LIN {X 0,Y 520.349,Z 992.129,A -85,B 0,C 180,E1 23655.766,E2 23655.766} C_VEL
LIN {X 0,Y 520.731,Z 981.899,A -85,B 0,C 180,E1 23653.265,E2 23653.265} C_VEL
LIN {X 0,Y 521.246,Z 970.85,A -85,B 0,C 180,E1 23650.972,E2 23650.972} C_VEL
LIN {X 0,Y 521.945,Z 957.785,A -85,B 0,C 180,E1 23648.66,E2 23648.66} C_VEL
LIN {X 0,Y 522.858,Z 943.405,A -85,B 0,C 180,E1 23646.447,E2 23646.447} C_VEL
LIN {X 0,Y 523.896,Z 928.063,A -85,B 0,C 180,E1 23644.403,E2 23644.403} C_VEL
LIN {X 0,Y 525.181,Z 910.163,A -85,B 0,C 180,E1 23642.325,E2 23642.325} C_VEL
LIN {X 0,Y 526.584,Z 891.955,A -85,B 0,C 180,E1 23640.485,E2 23640.485} C_VEL
LIN {X 0,Y 527.977,Z 872.898,A -85,B 0,C 180,E1 23638.832,E2 23638.832} C_VEL
LIN {X 0,Y 529.538,Z 851.806,A -85,B 0,C 180,E1 23637.256,E2 23637.256} C_VEL
LIN {X 0,Y 530.891,Z 831.896,A -85,B 0,C 180,E1 23635.994,E2 23635.994} C_VEL
LIN {X 0,Y 532.274,Z 810.352,A -85,B 0,C 180,E1 23634.853,E2 23634.853} C_VEL
LIN {X 0,Y 533.339,Z 791.103,A -85,B 0,C 180,E1 23634.01,E2 23634.01} C_VEL
LIN {X 0,Y 534.429,Z 767.307,A -85,B 0,C 180,E1 23633.184,E2 23633.184} C_VEL
LIN {X 0,Y 535.228,Z 746.145,A -85,B 0,C 180,E1 23632.64,E2 23632.64} C_VEL
LIN {X 0,Y 535.848,Z 714.251,A -85,B 0,C 180,E1 23632.088,E2 23632.088} C_VEL
LIN {X 0,Y 538.7,Z 503.39,A -85,B 0,C 180,E1 23628.756,E2 23628.756} C_VEL
LIN {X 0,Y 539.869,Z 409.939,A -85,B 0,C 180,E1 23627.231,E2 23627.231} C_VEL
LIN {X 0,Y 537.49,Z 399.108,A -85,B 0,C 180,E1 23626.805,E2 23626.805} C_VEL
LIN {X 0,Y 531.85,Z 390.278,A -85,B 0,C 180,E1 23626.056,E2 23626.056} C_VEL
LIN {X 0,Y 523.892,Z 373.784,A -85,B 0,C 180,E1 23623.835,E2 23623.835} C_VEL
LIN {X 0,Y 520.607,Z 366.647,A -85,B 0,C 180,E1 23622.814,E2 23622.814} C_VEL
LIN {X 0,Y 520.573,Z 366.184,A -85,B 0,C 180,E1 23622.24,E2 23622.24} C_VEL
LIN {X 0,Y 520.511,Z 366.188,A -85,B 0,C 180,E1 23619.054,E2 23619.054} C_VEL
LIN {X 0,Y 520.521,Z 366.183,A -85,B 0,C 180,E1 23615.593,E2 23615.593} C_VEL
LIN {X 0,Y 520.548,Z 366.206,A -85,B 0,C 180,E1 23612.323,E2 23612.323} C_VEL
LIN {X 0,Y 520.502,Z 366.203,A -85,B 0,C 180,E1 23609.078,E2 23609.078} C_VEL
LIN {X 0,Y 520.567,Z 366.201,A -85,B 0,C 180,E1 23605.849,E2 23605.849} C_VEL
LIN {X 0,Y 520.502,Z 366.206,A -85,B 0,C 180,E1 23602.593,E2 23602.593} C_VEL
LIN {X 0,Y 520.525,Z 366.208,A -85,B 0,C 180,E1 23599.175,E2 23599.175} C_VEL
LIN {X 0,Y 520.539,Z 366.208,A -85,B 0,C 180,E1 23595.942,E2 23595.942} C_VEL
LIN {X 0,Y 520.511,Z 366.206,A -85,B 0,C 180,E1 23592.649,E2 23592.649} C_VEL
LIN {X 0,Y 520.577,Z 366.201,A -85,B 0,C 180,E1 23589.396,E2 23589.396} C_VEL
LIN {X 0,Y 520.514,Z 366.205,A -85,B 0,C 180,E1 23586.175,E2 23586.175} C_VEL
LIN {X 0,Y 520.543,Z 366.199,A -85,B 0,C 180,E1 23582.752,E2 23582.752} C_VEL
LIN {X 0,Y 520.542,Z 366.207,A -85,B 0,C 180,E1 23579.559,E2 23579.559} C_VEL
LIN {X 0,Y 520.524,Z 366.203,A -85,B 0,C 180,E1 23576.145,E2 23576.145} C_VEL
LIN {X 0,Y 520.587,Z 366.197,A -85,B 0,C 180,E1 23572.828,E2 23572.828} C_VEL
LIN {X 0,Y 520.534,Z 366.206,A -85,B 0,C 180,E1 23569.485,E2 23569.485} C_VEL
LIN {X 0,Y 520.535,Z 366.202,A -85,B 0,C 180,E1 23565.993,E2 23565.993} C_VEL
LIN {X 0,Y 520.588,Z 366.199,A -85,B 0,C 180,E1 23562.642,E2 23562.642} C_VEL
LIN {X 0,Y 520.538,Z 366.205,A -85,B 0,C 180,E1 23559.283,E2 23559.283} C_VEL
LIN {X 0,Y 520.548,Z 366.2,A -85,B 0,C 180,E1 23555.822,E2 23555.822} C_VEL
LIN {X 0,Y 520.588,Z 366.199,A -85,B 0,C 180,E1 23552.427,E2 23552.427} C_VEL
LIN {X 0,Y 520.539,Z 366.203,A -85,B 0,C 180,E1 23549.145,E2 23549.145} C_VEL
LIN {X 0,Y 520.573,Z 366.197,A -85,B 0,C 180,E1 23545.752,E2 23545.752} C_VEL
LIN {X 0,Y 520.58,Z 366.2,A -85,B 0,C 180,E1 23542.3,E2 23542.3} C_VEL
LIN {X 0,Y 520.546,Z 366.2,A -85,B 0,C 180,E1 23538.935,E2 23538.935} C_VEL
LIN {X 0,Y 520.587,Z 366.201,A -85,B 0,C 180,E1 23537.815,E2 23537.815} C_VEL
LIN {X 0,Y 519.589,Z 366.322,A -85,B 0,C 180,E1 23536.968,E2 23536.968} C_VEL
LIN {X 0,Y 513.085,Z 367.141,A -85,B 0,C 180,E1 23534.524,E2 23534.524} C_VEL
LIN {X 0,Y 512.648,Z 367.189,A -85,B 0,C 180,E1 23533.965,E2 23533.965} C_VEL
LIN {X 0,Y 512.615,Z 367.191,A -85,B 0,C 180,E1 23530.474,E2 23530.474} C_VEL
LIN {X 0,Y 512.624,Z 367.189,A -85,B 0,C 180,E1 23526.898,E2 23526.898} C_VEL
LIN {X 0,Y 512.646,Z 367.172,A -85,B 0,C 180,E1 23523.408,E2 23523.408} C_VEL
LIN {X 0,Y 512.631,Z 367.178,A -85,B 0,C 180,E1 23519.949,E2 23519.949} C_VEL
LIN {X 0,Y 512.622,Z 367.192,A -85,B 0,C 180,E1 23516.4,E2 23516.4} C_VEL
LIN {X 0,Y 512.647,Z 367.191,A -85,B 0,C 180,E1 23512.955,E2 23512.955} C_VEL
LIN {X 0,Y 512.645,Z 367.193,A -85,B 0,C 180,E1 23509.359,E2 23509.359} C_VEL
LIN {X 0,Y 512.648,Z 367.36,A -85,B 0,C 180,E1 23508.032,E2 23508.032} C_VEL
LIN {X 0,Y 513.024,Z 368.847,A -85,B 0,C 180,E1 23507.813,E2 23507.813} C_VEL
LIN {X 0,Y 514.992,Z 371.888,A -85,B 0,C 180,E1 23507.522,E2 23507.522} C_VEL
LIN {X 0,Y 516.385,Z 373.399,A -85,B 0,C 180,E1 23507.333,E2 23507.333} C_VEL
LIN {X 0,Y 519.013,Z 377.291,A -85,B 0,C 180,E1 23506.963,E2 23506.963} C_VEL
LIN {X 0,Y 530.622,Z 393.994,A -85,B 0,C 180,E1 23505.404,E2 23505.404} C_VEL
LIN {X 0,Y 533.879,Z 399.167,A -85,B 0,C 180,E1 23504.979,E2 23504.979} C_VEL
LIN {X 0,Y 530.564,Z 613.236,A -85,B 0,C 180,E1 23501.524,E2 23501.524} C_VEL
LIN {X 0,Y 529.036,Z 711.437,A -85,B 0,C 180,E1 23499.944,E2 23499.944} C_VEL
LIN {X 0,Y 528.194,Z 733.986,A -85,B 0,C 180,E1 23499.396,E2 23499.396} C_VEL
LIN {X 0,Y 527.019,Z 757.223,A -85,B 0,C 180,E1 23498.623,E2 23498.623} C_VEL
LIN {X 0,Y 525.744,Z 778.536,A -85,B 0,C 180,E1 23497.702,E2 23497.702} C_VEL
LIN {X 0,Y 524.274,Z 800.078,A -85,B 0,C 180,E1 23496.567,E2 23496.567} C_VEL
LIN {X 0,Y 522.652,Z 821.532,A -85,B 0,C 180,E1 23495.21,E2 23495.21} C_VEL
LIN {X 0,Y 520.974,Z 842.55,A -85,B 0,C 180,E1 23493.628,E2 23493.628} C_VEL
LIN {X 0,Y 519.313,Z 862.459,A -85,B 0,C 180,E1 23491.872,E2 23491.872} C_VEL
LIN {X 0,Y 517.78,Z 880.735,A -85,B 0,C 180,E1 23489.997,E2 23489.997} C_VEL
LIN {X 0,Y 516.352,Z 898.567,A -85,B 0,C 180,E1 23487.888,E2 23487.888} C_VEL
LIN {X 0,Y 515.122,Z 914.905,A -85,B 0,C 180,E1 23485.655,E2 23485.655} C_VEL
LIN {X 0,Y 514.093,Z 929.824,A -85,B 0,C 180,E1 23483.296,E2 23483.296} C_VEL
LIN {X 0,Y 513.292,Z 943.254,A -85,B 0,C 180,E1 23480.806,E2 23480.806} C_VEL
LIN {X 0,Y 512.729,Z 954.794,A -85,B 0,C 180,E1 23478.296,E2 23478.296} C_VEL
LIN {X 0,Y 512.352,Z 964.036,A -85,B 0,C 180,E1 23475.878,E2 23475.878} C_VEL
LIN {X 0,Y 512.081,Z 972.48,A -85,B 0,C 180,E1 23473.201,E2 23473.201} C_VEL
LIN {X 0,Y 511.963,Z 978.61,A -85,B 0,C 180,E1 23470.725,E2 23470.725} C_VEL
LIN {X 0,Y 511.913,Z 983.402,A -85,B 0,C 180,E1 23468.09,E2 23468.09} C_VEL
LIN {X 0,Y 511.915,Z 986.412,A -85,B 0,C 180,E1 23465.531,E2 23465.531} C_VEL
LIN {X 0,Y 511.903,Z 987.824,A -85,B 0,C 180,E1 23462.926,E2 23462.926} C_VEL
LIN {X 0,Y 511.9,Z 987.73,A -85,B 0,C 180,E1 23460.511,E2 23460.511} C_VEL
LIN {X 0,Y 511.908,Z 986.022,A -85,B 0,C 180,E1 23457.962,E2 23457.962} C_VEL
LIN {X 0,Y 511.933,Z 982.695,A -85,B 0,C 180,E1 23455.362,E2 23455.362} C_VEL
LIN {X 0,Y 511.996,Z 977.795,A -85,B 0,C 180,E1 23452.823,E2 23452.823} C_VEL
LIN {X 0,Y 512.141,Z 971.297,A -85,B 0,C 180,E1 23450.284,E2 23450.284} C_VEL
LIN {X 0,Y 512.374,Z 963.32,A -85,B 0,C 180,E1 23447.831,E2 23447.831} C_VEL
LIN {X 0,Y 512.764,Z 953.763,A -85,B 0,C 180,E1 23445.376,E2 23445.376} C_VEL
LIN {X 0,Y 513.339,Z 942.306,A -85,B 0,C 180,E1 23442.913,E2 23442.913} C_VEL
LIN {X 0,Y 514.168,Z 928.617,A -85,B 0,C 180,E1 23440.411,E2 23440.411} C_VEL
LIN {X 0,Y 515.189,Z 913.932,A -85,B 0,C 180,E1 23438.11,E2 23438.11} C_VEL
LIN {X 0,Y 516.424,Z 897.762,A -85,B 0,C 180,E1 23435.92,E2 23435.92} C_VEL
LIN {X 0,Y 517.885,Z 879.526,A -85,B 0,C 180,E1 23433.782,E2 23433.782} C_VEL
LIN {X 0,Y 519.416,Z 861.022,A -85,B 0,C 180,E1 23431.904,E2 23431.904} C_VEL
LIN {X 0,Y 521.084,Z 841.323,A -85,B 0,C 180,E1 23430.181,E2 23430.181} C_VEL
LIN {X 0,Y 522.756,Z 820.167,A -85,B 0,C 180,E1 23428.605,E2 23428.605} C_VEL
LIN {X 0,Y 524.336,Z 799.285,A -85,B 0,C 180,E1 23427.297,E2 23427.297} C_VEL
LIN {X 0,Y 525.804,Z 777.515,A -85,B 0,C 180,E1 23426.16,E2 23426.16} C_VEL
LIN {X 0,Y 527.123,Z 755.205,A -85,B 0,C 180,E1 23425.214,E2 23425.214} C_VEL
LIN {X 0,Y 528.261,Z 732.587,A -85,B 0,C 180,E1 23424.473,E2 23424.473} C_VEL
LIN {X 0,Y 529.086,Z 709.622,A -85,B 0,C 180,E1 23423.929,E2 23423.929} C_VEL
LIN {X 0,Y 532.283,Z 499.238,A -85,B 0,C 180,E1 23420.56,E2 23420.56} C_VEL
LIN {X 0,Y 533.734,Z 398.668,A -85,B 0,C 180,E1 23418.906,E2 23418.906} C_VEL
LIN {X 0,Y 524.824,Z 385.59,A -85,B 0,C 180,E1 23417.734,E2 23417.734} C_VEL
LIN {X 0,Y 519.029,Z 377.339,A -85,B 0,C 180,E1 23416.94,E2 23416.94} C_VEL
LIN {X 0,Y 516.307,Z 373.278,A -85,B 0,C 180,E1 23416.554,E2 23416.554} C_VEL
LIN {X 0,Y 513.441,Z 369.804,A -85,B 0,C 180,E1 23416.154,E2 23416.154} C_VEL
LIN {X 0,Y 512.74,Z 367.777,A -85,B 0,C 180,E1 23415.96,E2 23415.96} C_VEL
LIN {X 0,Y 512.647,Z 367.178,A -85,B 0,C 180,E1 23415.614,E2 23415.614} C_VEL
LIN {X 0,Y 512.643,Z 367.188,A -85,B 0,C 180,E1 23412.046,E2 23412.046} C_VEL
LIN {X 0,Y 512.634,Z 367.194,A -85,B 0,C 180,E1 23408.525,E2 23408.525} C_VEL
LIN {X 0,Y 512.641,Z 367.184,A -85,B 0,C 180,E1 23405.036,E2 23405.036} C_VEL
LIN {X 0,Y 512.631,Z 367.193,A -85,B 0,C 180,E1 23401.565,E2 23401.565} C_VEL
LIN {X 0,Y 512.644,Z 367.19,A -85,B 0,C 180,E1 23398.1,E2 23398.1} C_VEL
LIN {X 0,Y 512.642,Z 367.186,A -85,B 0,C 180,E1 23394.516,E2 23394.516} C_VEL
LIN {X 0,Y 512.622,Z 367.191,A -85,B 0,C 180,E1 23391.137,E2 23391.137} C_VEL
LIN {X 0,Y 512.622,Z 367.194,A -85,B 0,C 180,E1 23387.611,E2 23387.611} C_VEL
LIN {X 0,Y 512.648,Z 367.191,A -85,B 0,C 180,E1 23384.154,E2 23384.154} C_VEL
LIN {X 0,Y 512.616,Z 367.192,A -85,B 0,C 180,E1 23380.746,E2 23380.746} C_VEL
LIN {X 0,Y 512.601,Z 367.193,A -85,B 0,C 180,E1 23377.282,E2 23377.282} C_VEL
LIN {X 0,Y 512.647,Z 367.187,A -85,B 0,C 180,E1 23373.971,E2 23373.971} C_VEL
LIN {X 0,Y 512.588,Z 367.189,A -85,B 0,C 180,E1 23370.686,E2 23370.686} C_VEL
LIN {X 0,Y 512.587,Z 367.199,A -85,B 0,C 180,E1 23367.162,E2 23367.162} C_VEL
LIN {X 0,Y 512.63,Z 367.19,A -85,B 0,C 180,E1 23363.854,E2 23363.854} C_VEL
LIN {X 0,Y 512.567,Z 367.202,A -85,B 0,C 180,E1 23360.512,E2 23360.512} C_VEL
LIN {X 0,Y 512.633,Z 367.461,A -85,B 0,C 180,E1 23358,E2 23358} C_VEL
LIN {X 0,Y 514.255,Z 371.158,A -85,B 0,C 180,E1 23357.421,E2 23357.421} C_VEL
LIN {X 0,Y 522.336,Z 388.024,A -85,B 0,C 180,E1 23355.063,E2 23355.063} C_VEL
LIN {X 0,Y 524.102,Z 391.266,A -85,B 0,C 180,E1 23354.714,E2 23354.714} C_VEL
LIN {X 0,Y 532.473,Z 404.496,A -85,B 0,C 180,E1 23353.596,E2 23353.596} C_VEL
LIN {X 0,Y 534.057,Z 413.512,A -85,B 0,C 180,E1 23353.272,E2 23353.272} C_VEL
LIN {X 0,Y 530.901,Z 620.252,A -85,B 0,C 180,E1 23349.935,E2 23349.935} C_VEL
LIN {X 0,Y 529.048,Z 740.56,A -85,B 0,C 180,E1 23348.004,E2 23348.004} C_VEL
LIN {X 0,Y 528.187,Z 763.41,A -85,B 0,C 180,E1 23347.452,E2 23347.452} C_VEL
LIN {X 0,Y 527.178,Z 784.187,A -85,B 0,C 180,E1 23346.778,E2 23346.778} C_VEL
LIN {X 0,Y 525.864,Z 806.34,A -85,B 0,C 180,E1 23345.849,E2 23345.849} C_VEL
LIN {X 0,Y 524.54,Z 826.536,A -85,B 0,C 180,E1 23344.815,E2 23344.815} C_VEL
LIN {X 0,Y 522.895,Z 848.102,A -85,B 0,C 180,E1 23343.483,E2 23343.483} C_VEL
LIN {X 0,Y 521.357,Z 867.974,A -85,B 0,C 180,E1 23342.042,E2 23342.042} C_VEL
LIN {X 0,Y 519.726,Z 887.242,A -85,B 0,C 180,E1 23340.398,E2 23340.398} C_VEL
LIN {X 0,Y 518.112,Z 906.765,A -85,B 0,C 180,E1 23338.47,E2 23338.47} C_VEL
LIN {X 0,Y 516.731,Z 923.638,A -85,B 0,C 180,E1 23336.553,E2 23336.553} C_VEL
LIN {X 0,Y 515.543,Z 939.127,A -85,B 0,C 180,E1 23334.524,E2 23334.524} C_VEL
LIN {X 0,Y 514.479,Z 954.204,A -85,B 0,C 180,E1 23332.273,E2 23332.273} C_VEL
LIN {X 0,Y 513.631,Z 967.075,A -85,B 0,C 180,E1 23330.039,E2 23330.039} C_VEL
LIN {X 0,Y 512.948,Z 979.793,A -85,B 0,C 180,E1 23327.471,E2 23327.471} C_VEL
LIN {X 0,Y 512.523,Z 989.518,A -85,B 0,C 180,E1 23325.157,E2 23325.157} C_VEL
LIN {X 0,Y 512.205,Z 998.524,A -85,B 0,C 180,E1 23322.571,E2 23322.571} C_VEL
LIN {X 0,Y 512.027,Z 1005.249,A -85,B 0,C 180,E1 23320.206,E2 23320.206} C_VEL
LIN {X 0,Y 511.953,Z 1010.629,A -85,B 0,C 180,E1 23317.748,E2 23317.748} C_VEL
LIN {X 0,Y 511.91,Z 1014.273,A -85,B 0,C 180,E1 23315.495,E2 23315.495} C_VEL
LIN {X 0,Y 511.89,Z 1016.917,A -85,B 0,C 180,E1 23312.914,E2 23312.914} C_VEL
LIN {X 0,Y 511.883,Z 1017.872,A -85,B 0,C 180,E1 23310.675,E2 23310.675} C_VEL
LIN {X 0,Y 511.909,Z 1017.528,A -85,B 0,C 180,E1 23308.101,E2 23308.101} C_VEL
LIN {X 0,Y 511.911,Z 1015.733,A -85,B 0,C 180,E1 23305.747,E2 23305.747} C_VEL
LIN {X 0,Y 511.925,Z 1012.5,A -85,B 0,C 180,E1 23303.274,E2 23303.274} C_VEL
LIN {X 0,Y 511.996,Z 1007.837,A -85,B 0,C 180,E1 23300.902,E2 23300.902} C_VEL
LIN {X 0,Y 512.119,Z 1001.528,A -85,B 0,C 180,E1 23298.403,E2 23298.403} C_VEL
LIN {X 0,Y 512.355,Z 993.422,A -85,B 0,C 180,E1 23295.903,E2 23295.903} C_VEL
LIN {X 0,Y 512.746,Z 983.956,A -85,B 0,C 180,E1 23293.463,E2 23293.463} C_VEL
LIN {X 0,Y 513.275,Z 973.174,A -85,B 0,C 180,E1 23291.138,E2 23291.138} C_VEL
LIN {X 0,Y 514.072,Z 959.885,A -85,B 0,C 180,E1 23288.676,E2 23288.676} C_VEL
LIN {X 0,Y 514.991,Z 946.596,A -85,B 0,C 180,E1 23286.551,E2 23286.551} C_VEL
LIN {X 0,Y 516.168,Z 930.762,A -85,B 0,C 180,E1 23284.351,E2 23284.351} C_VEL
LIN {X 0,Y 517.52,Z 914.034,A -85,B 0,C 180,E1 23282.317,E2 23282.317} C_VEL
LIN {X 0,Y 518.986,Z 896.227,A -85,B 0,C 180,E1 23280.454,E2 23280.454} C_VEL
LIN {X 0,Y 520.627,Z 876.321,A -85,B 0,C 180,E1 23278.643,E2 23278.643} C_VEL
LIN {X 0,Y 522.234,Z 856.967,A -85,B 0,C 180,E1 23277.132,E2 23277.132} C_VEL
LIN {X 0,Y 523.815,Z 835.912,A -85,B 0,C 180,E1 23275.735,E2 23275.735} C_VEL
LIN {X 0,Y 525.403,Z 814.179,A -85,B 0,C 180,E1 23274.525,E2 23274.525} C_VEL
LIN {X 0,Y 526.667,Z 793.392,A -85,B 0,C 180,E1 23273.586,E2 23273.586} C_VEL
LIN {X 0,Y 527.825,Z 771.737,A -85,B 0,C 180,E1 23272.79,E2 23272.79} C_VEL
LIN {X 0,Y 528.721,Z 749.391,A -85,B 0,C 180,E1 23272.186,E2 23272.186} C_VEL
LIN {X 0,Y 529.41,Z 723.55,A -85,B 0,C 180,E1 23271.701,E2 23271.701} C_VEL
LIN {X 0,Y 532.519,Z 513.255,A -85,B 0,C 180,E1 23268.347,E2 23268.347} C_VEL
LIN {X 0,Y 533.929,Z 411.728,A -85,B 0,C 180,E1 23266.678,E2 23266.678} C_VEL
LIN {X 0,Y 532.159,Z 403.642,A -85,B 0,C 180,E1 23266.352,E2 23266.352} C_VEL
LIN {X 0,Y 523.281,Z 389.92,A -85,B 0,C 180,E1 23265.144,E2 23265.144} C_VEL
LIN {X 0,Y 516.26,Z 375.275,A -85,B 0,C 180,E1 23263.108,E2 23263.108} C_VEL
LIN {X 0,Y 512.665,Z 367.588,A -85,B 0,C 180,E1 23261.958,E2 23261.958} C_VEL
LIN {X 0,Y 512.577,Z 367.19,A -85,B 0,C 180,E1 23261.099,E2 23261.099} C_VEL
LIN {X 0,Y 512.585,Z 367.2,A -85,B 0,C 180,E1 23257.628,E2 23257.628} C_VEL
LIN {X 0,Y 512.616,Z 367.174,A -85,B 0,C 180,E1 23254.311,E2 23254.311} C_VEL
LIN {X 0,Y 512.563,Z 367.176,A -85,B 0,C 180,E1 23250.996,E2 23250.996} C_VEL
LIN {X 0,Y 512.608,Z 367.197,A -85,B 0,C 180,E1 23247.66,E2 23247.66} C_VEL
LIN {X 0,Y 512.578,Z 367.199,A -85,B 0,C 180,E1 23244.376,E2 23244.376} C_VEL
LIN {X 0,Y 512.566,Z 367.194,A -85,B 0,C 180,E1 23240.887,E2 23240.887} C_VEL
LIN {X 0,Y 512.632,Z 367.19,A -85,B 0,C 180,E1 23237.596,E2 23237.596} C_VEL
LIN {X 0,Y 512.571,Z 367.191,A -85,B 0,C 180,E1 23234.343,E2 23234.343} C_VEL
LIN {X 0,Y 512.589,Z 367.195,A -85,B 0,C 180,E1 23230.906,E2 23230.906} C_VEL
LIN {X 0,Y 512.614,Z 367.191,A -85,B 0,C 180,E1 23227.621,E2 23227.621} C_VEL
LIN {X 0,Y 512.576,Z 367.194,A -85,B 0,C 180,E1 23224.25,E2 23224.25} C_VEL
LIN {X 0,Y 512.627,Z 367.193,A -85,B 0,C 180,E1 23220.894,E2 23220.894} C_VEL
LIN {X 0,Y 512.594,Z 367.193,A -85,B 0,C 180,E1 23217.652,E2 23217.652} C_VEL
LIN {X 0,Y 512.587,Z 367.194,A -85,B 0,C 180,E1 23214.106,E2 23214.106} C_VEL
LIN {X 0,Y 512.648,Z 367.193,A -85,B 0,C 180,E1 23210.797,E2 23210.797} C_VEL
LIN {X 0,Y 512.593,Z 367.192,A -85,B 0,C 180,E1 23207.495,E2 23207.495} C_VEL
LIN {X 0,Y 512.597,Z 367.192,A -85,B 0,C 180,E1 23203.919,E2 23203.919} C_VEL
LIN {X 0,Y 512.65,Z 367.192,A -85,B 0,C 180,E1 23200.517,E2 23200.517} C_VEL
LIN {X 0,Y 512.603,Z 367.191,A -85,B 0,C 180,E1 23197.159,E2 23197.159} C_VEL
LIN {X 0,Y 512.604,Z 367.191,A -85,B 0,C 180,E1 23193.594,E2 23193.594} C_VEL
LIN {X 0,Y 512.652,Z 367.19,A -85,B 0,C 180,E1 23190.175,E2 23190.175} C_VEL
LIN {X 0,Y 512.613,Z 367.193,A -85,B 0,C 180,E1 23186.763,E2 23186.763} C_VEL
LIN {X 0,Y 512.608,Z 367.192,A -85,B 0,C 180,E1 23183.214,E2 23183.214} C_VEL
LIN {X 0,Y 512.651,Z 367.186,A -85,B 0,C 180,E1 23179.791,E2 23179.791} C_VEL
LIN {X 0,Y 512.628,Z 367.191,A -85,B 0,C 180,E1 23176.333,E2 23176.333} C_VEL
LIN {X 0,Y 512.648,Z 367.189,A -85,B 0,C 180,E1 23173.965,E2 23173.965} C_VEL
LIN {X 0,Y 511.649,Z 367.308,A -85,B 0,C 180,E1 23173.104,E2 23173.104} C_VEL
LIN {X 0,Y 505.207,Z 368.114,A -85,B 0,C 180,E1 23170.684,E2 23170.684} C_VEL
LIN {X 0,Y 504.699,Z 368.177,A -85,B 0,C 180,E1 23170.054,E2 23170.054} C_VEL
LIN {X 0,Y 504.676,Z 368.181,A -85,B 0,C 180,E1 23166.602,E2 23166.602} C_VEL
LIN {X 0,Y 504.703,Z 368.163,A -85,B 0,C 180,E1 23163.07,E2 23163.07} C_VEL
LIN {X 0,Y 504.707,Z 368.158,A -85,B 0,C 180,E1 23159.551,E2 23159.551} C_VEL
LIN {X 0,Y 504.683,Z 368.173,A -85,B 0,C 180,E1 23156.087,E2 23156.087} C_VEL
LIN {X 0,Y 504.692,Z 368.177,A -85,B 0,C 180,E1 23152.475,E2 23152.475} C_VEL
LIN {X 0,Y 504.721,Z 368.305,A -85,B 0,C 180,E1 23148.979,E2 23148.979} C_VEL
LIN {X 0,Y 505.081,Z 369.781,A -85,B 0,C 180,E1 23148.738,E2 23148.738} C_VEL
LIN {X 0,Y 507.099,Z 372.938,A -85,B 0,C 180,E1 23148.424,E2 23148.424} C_VEL
LIN {X 0,Y 508.553,Z 374.512,A -85,B 0,C 180,E1 23148.219,E2 23148.219} C_VEL
LIN {X 0,Y 511.228,Z 378.407,A -85,B 0,C 180,E1 23147.826,E2 23147.826} C_VEL
LIN {X 0,Y 522.821,Z 394.818,A -85,B 0,C 180,E1 23146.209,E2 23146.209} C_VEL
LIN {X 0,Y 527.98,Z 402.563,A -85,B 0,C 180,E1 23145.518,E2 23145.518} C_VEL
LIN {X 0,Y 524.318,Z 618.399,A -85,B 0,C 180,E1 23142,E2 23142} C_VEL
LIN {X 0,Y 522.728,Z 711.407,A -85,B 0,C 180,E1 23140.487,E2 23140.487} C_VEL
LIN {X 0,Y 521.821,Z 734.028,A -85,B 0,C 180,E1 23139.933,E2 23139.933} C_VEL
LIN {X 0,Y 520.548,Z 757.204,A -85,B 0,C 180,E1 23139.156,E2 23139.156} C_VEL
LIN {X 0,Y 519.106,Z 779.291,A -85,B 0,C 180,E1 23138.191,E2 23138.191} C_VEL
LIN {X 0,Y 517.507,Z 800.717,A -85,B 0,C 180,E1 23137.043,E2 23137.043} C_VEL
LIN {X 0,Y 515.798,Z 821.334,A -85,B 0,C 180,E1 23135.726,E2 23135.726} C_VEL
LIN {X 0,Y 513.968,Z 842.409,A -85,B 0,C 180,E1 23134.124,E2 23134.124} C_VEL
LIN {X 0,Y 512.172,Z 861.761,A -85,B 0,C 180,E1 23132.402,E2 23132.402} C_VEL
LIN {X 0,Y 510.506,Z 880.135,A -85,B 0,C 180,E1 23130.502,E2 23130.502} C_VEL
LIN {X 0,Y 508.942,Z 897.623,A -85,B 0,C 180,E1 23128.421,E2 23128.421} C_VEL
LIN {X 0,Y 507.621,Z 913.339,A -85,B 0,C 180,E1 23126.27,E2 23126.27} C_VEL
LIN {X 0,Y 506.47,Z 928.424,A -85,B 0,C 180,E1 23123.877,E2 23123.877} C_VEL
LIN {X 0,Y 505.545,Z 942.067,A -85,B 0,C 180,E1 23121.352,E2 23121.352} C_VEL
LIN {X 0,Y 504.9,Z 953.235,A -85,B 0,C 180,E1 23118.922,E2 23118.922} C_VEL
LIN {X 0,Y 504.44,Z 963.155,A -85,B 0,C 180,E1 23116.354,E2 23116.354} C_VEL
LIN {X 0,Y 504.168,Z 971.121,A -85,B 0,C 180,E1 23113.877,E2 23113.877} C_VEL
LIN {X 0,Y 504.013,Z 977.756,A -85,B 0,C 180,E1 23111.251,E2 23111.251} C_VEL
LIN {X 0,Y 503.935,Z 982.605,A -85,B 0,C 180,E1 23108.707,E2 23108.707} C_VEL
LIN {X 0,Y 503.896,Z 985.917,A -85,B 0,C 180,E1 23106.119,E2 23106.119} C_VEL
LIN {X 0,Y 503.889,Z 987.674,A -85,B 0,C 180,E1 23103.607,E2 23103.607} C_VEL
LIN {X 0,Y 503.913,Z 987.841,A -85,B 0,C 180,E1 23101.049,E2 23101.049} C_VEL
LIN {X 0,Y 503.907,Z 986.433,A -85,B 0,C 180,E1 23098.346,E2 23098.346} C_VEL
LIN {X 0,Y 503.908,Z 983.561,A -85,B 0,C 180,E1 23095.835,E2 23095.835} C_VEL
LIN {X 0,Y 503.962,Z 979.096,A -85,B 0,C 180,E1 23093.278,E2 23093.278} C_VEL
LIN {X 0,Y 504.111,Z 972.871,A -85,B 0,C 180,E1 23090.673,E2 23090.673} C_VEL
LIN {X 0,Y 504.395,Z 964.46,A -85,B 0,C 180,E1 23087.929,E2 23087.929} C_VEL
LIN {X 0,Y 504.797,Z 955.293,A -85,B 0,C 180,E1 23085.476,E2 23085.476} C_VEL
LIN {X 0,Y 505.411,Z 943.967,A -85,B 0,C 180,E1 23082.945,E2 23082.945} C_VEL
LIN {X 0,Y 506.255,Z 931.103,A -85,B 0,C 180,E1 23080.5,E2 23080.5} C_VEL
LIN {X 0,Y 507.388,Z 916.279,A -85,B 0,C 180,E1 23078.083,E2 23078.083} C_VEL
LIN {X 0,Y 508.716,Z 900.445,A -85,B 0,C 180,E1 23075.853,E2 23075.853} C_VEL
LIN {X 0,Y 510.219,Z 883.315,A -85,B 0,C 180,E1 23073.757,E2 23073.757} C_VEL
LIN {X 0,Y 511.897,Z 864.989,A -85,B 0,C 180,E1 23071.822,E2 23071.822} C_VEL
LIN {X 0,Y 513.624,Z 845.937,A -85,B 0,C 180,E1 23070.084,E2 23070.084} C_VEL
LIN {X 0,Y 515.422,Z 825.761,A -85,B 0,C 180,E1 23068.503,E2 23068.503} C_VEL
LIN {X 0,Y 517.119,Z 805.535,A -85,B 0,C 180,E1 23067.15,E2 23067.15} C_VEL
LIN {X 0,Y 518.871,Z 783.109,A -85,B 0,C 180,E1 23065.903,E2 23065.903} C_VEL
LIN {X 0,Y 520.253,Z 761.88,A -85,B 0,C 180,E1 23064.946,E2 23064.946} C_VEL
LIN {X 0,Y 521.581,Z 738.114,A -85,B 0,C 180,E1 23064.1,E2 23064.1} C_VEL
LIN {X 0,Y 522.579,Z 715.323,A -85,B 0,C 180,E1 23063.508,E2 23063.508} C_VEL
LIN {X 0,Y 523.313,Z 682.027,A -85,B 0,C 180,E1 23062.927,E2 23062.927} C_VEL
LIN {X 0,Y 526.759,Z 472.174,A -85,B 0,C 180,E1 23059.538,E2 23059.538} C_VEL
LIN {X 0,Y 527.895,Z 402.246,A -85,B 0,C 180,E1 23058.372,E2 23058.372} C_VEL
LIN {X 0,Y 515.015,Z 383.608,A -85,B 0,C 180,E1 23056.612,E2 23056.612} C_VEL
LIN {X 0,Y 510.873,Z 378.049,A -85,B 0,C 180,E1 23056.02,E2 23056.02} C_VEL
LIN {X 0,Y 507.824,Z 373.56,A -85,B 0,C 180,E1 23055.561,E2 23055.561} C_VEL
LIN {X 0,Y 505.444,Z 370.693,A -85,B 0,C 180,E1 23055.21,E2 23055.21} C_VEL
LIN {X 0,Y 504.804,Z 368.876,A -85,B 0,C 180,E1 23055.039,E2 23055.039} C_VEL
LIN {X 0,Y 504.683,Z 368.168,A -85,B 0,C 180,E1 23054.69,E2 23054.69} C_VEL
LIN {X 0,Y 504.699,Z 368.178,A -85,B 0,C 180,E1 23051.195,E2 23051.195} C_VEL
LIN {X 0,Y 504.698,Z 368.176,A -85,B 0,C 180,E1 23047.743,E2 23047.743} C_VEL
LIN {X 0,Y 504.703,Z 368.18,A -85,B 0,C 180,E1 23044.204,E2 23044.204} C_VEL
LIN {X 0,Y 504.7,Z 368.18,A -85,B 0,C 180,E1 23040.682,E2 23040.682} C_VEL
LIN {X 0,Y 504.694,Z 368.172,A -85,B 0,C 180,E1 23037.162,E2 23037.162} C_VEL
LIN {X 0,Y 504.687,Z 368.181,A -85,B 0,C 180,E1 23033.631,E2 23033.631} C_VEL
LIN {X 0,Y 504.707,Z 368.18,A -85,B 0,C 180,E1 23030.191,E2 23030.191} C_VEL
LIN {X 0,Y 504.696,Z 368.179,A -85,B 0,C 180,E1 23026.715,E2 23026.715} C_VEL
LIN {X 0,Y 504.669,Z 368.182,A -85,B 0,C 180,E1 23023.306,E2 23023.306} C_VEL
LIN {X 0,Y 504.701,Z 368.176,A -85,B 0,C 180,E1 23019.836,E2 23019.836} C_VEL
LIN {X 0,Y 504.687,Z 368.176,A -85,B 0,C 180,E1 23016.41,E2 23016.41} C_VEL
LIN {X 0,Y 504.652,Z 368.182,A -85,B 0,C 180,E1 23013.018,E2 23013.018} C_VEL
LIN {X 0,Y 504.692,Z 368.183,A -85,B 0,C 180,E1 23009.657,E2 23009.657} C_VEL
LIN {X 0,Y 504.658,Z 368.185,A -85,B 0,C 180,E1 23006.307,E2 23006.307} C_VEL
LIN {X 0,Y 504.632,Z 368.188,A -85,B 0,C 180,E1 23002.821,E2 23002.821} C_VEL
LIN {X 0,Y 504.678,Z 368.179,A -85,B 0,C 180,E1 22999.472,E2 22999.472} C_VEL
LIN {X 0,Y 504.699,Z 368.65,A -85,B 0,C 180,E1 22998.829,E2 22998.829} C_VEL
LIN {X 0,Y 506.28,Z 372.154,A -85,B 0,C 180,E1 22998.276,E2 22998.276} C_VEL
LIN {X 0,Y 513.096,Z 386.032,A -85,B 0,C 180,E1 22996.229,E2 22996.229} C_VEL
LIN {X 0,Y 515.022,Z 389.931,A -85,B 0,C 180,E1 22995.74,E2 22995.74} C_VEL
LIN {X 0,Y 527.078,Z 408.684,A -85,B 0,C 180,E1 22994.071,E2 22994.071} C_VEL
LIN {X 0,Y 528.168,Z 415.327,A -85,B 0,C 180,E1 22993.835,E2 22993.835} C_VEL
LIN {X 0,Y 524.719,Z 623.112,A -85,B 0,C 180,E1 22990.451,E2 22990.451} C_VEL
LIN {X 0,Y 522.742,Z 740.56,A -85,B 0,C 180,E1 22988.546,E2 22988.546} C_VEL
LIN {X 0,Y 521.82,Z 763.278,A -85,B 0,C 180,E1 22987.994,E2 22987.994} C_VEL
LIN {X 0,Y 520.768,Z 783.428,A -85,B 0,C 180,E1 22987.337,E2 22987.337} C_VEL
LIN {X 0,Y 519.282,Z 806.337,A -85,B 0,C 180,E1 22986.376,E2 22986.376} C_VEL
LIN {X 0,Y 517.77,Z 827.658,A -85,B 0,C 180,E1 22985.27,E2 22985.27} C_VEL
LIN {X 0,Y 516.052,Z 848.221,A -85,B 0,C 180,E1 22983.978,E2 22983.978} C_VEL
LIN {X 0,Y 514.336,Z 868.226,A -85,B 0,C 180,E1 22982.51,E2 22982.51} C_VEL
LIN {X 0,Y 512.591,Z 887.24,A -85,B 0,C 180,E1 22980.867,E2 22980.867} C_VEL
LIN {X 0,Y 510.802,Z 906.763,A -85,B 0,C 180,E1 22978.916,E2 22978.916} C_VEL
LIN {X 0,Y 509.334,Z 923.13,A -85,B 0,C 180,E1 22977.032,E2 22977.032} C_VEL
LIN {X 0,Y 507.971,Z 939.125,A -85,B 0,C 180,E1 22974.915,E2 22974.915} C_VEL
LIN {X 0,Y 506.778,Z 954.206,A -85,B 0,C 180,E1 22972.63,E2 22972.63} C_VEL
LIN {X 0,Y 505.846,Z 967.073,A -85,B 0,C 180,E1 22970.361,E2 22970.361} C_VEL
LIN {X 0,Y 505.09,Z 979.613,A -85,B 0,C 180,E1 22967.794,E2 22967.794} C_VEL
LIN {X 0,Y 504.598,Z 989.517,A -85,B 0,C 180,E1 22965.401,E2 22965.401} C_VEL
LIN {X 0,Y 504.253,Z 998.337,A -85,B 0,C 180,E1 22962.834,E2 22962.834} C_VEL
LIN {X 0,Y 504.067,Z 1004.858,A -85,B 0,C 180,E1 22960.518,E2 22960.518} C_VEL
LIN {X 0,Y 503.967,Z 1010.629,A -85,B 0,C 180,E1 22957.871,E2 22957.871} C_VEL
LIN {X 0,Y 503.912,Z 1014.432,A -85,B 0,C 180,E1 22955.468,E2 22955.468} C_VEL
LIN {X 0,Y 503.895,Z 1016.985,A -85,B 0,C 180,E1 22952.847,E2 22952.847} C_VEL
LIN {X 0,Y 503.884,Z 1017.894,A -85,B 0,C 180,E1 22950.572,E2 22950.572} C_VEL
LIN {X 0,Y 503.914,Z 1017.394,A -85,B 0,C 180,E1 22947.843,E2 22947.843} C_VEL
LIN {X 0,Y 503.905,Z 1015.505,A -85,B 0,C 180,E1 22945.451,E2 22945.451} C_VEL
LIN {X 0,Y 503.919,Z 1011.807,A -85,B 0,C 180,E1 22942.782,E2 22942.782} C_VEL
LIN {X 0,Y 504,Z 1007.327,A -85,B 0,C 180,E1 22940.526,E2 22940.526} C_VEL
LIN {X 0,Y 504.182,Z 1000.48,A -85,B 0,C 180,E1 22937.869,E2 22937.869} C_VEL
LIN {X 0,Y 504.445,Z 992.949,A -85,B 0,C 180,E1 22935.542,E2 22935.542} C_VEL
LIN {X 0,Y 504.913,Z 982.926,A -85,B 0,C 180,E1 22932.962,E2 22932.962} C_VEL
LIN {X 0,Y 505.539,Z 972.015,A -85,B 0,C 180,E1 22930.598,E2 22930.598} C_VEL
LIN {X 0,Y 506.454,Z 958.482,A -85,B 0,C 180,E1 22928.096,E2 22928.096} C_VEL
LIN {X 0,Y 507.573,Z 944.064,A -85,B 0,C 180,E1 22925.79,E2 22925.79} C_VEL
LIN {X 0,Y 508.88,Z 928.361,A -85,B 0,C 180,E1 22923.631,E2 22923.631} C_VEL
LIN {X 0,Y 510.5,Z 910.161,A -85,B 0,C 180,E1 22921.457,E2 22921.457} C_VEL
LIN {X 0,Y 512.149,Z 892.227,A -85,B 0,C 180,E1 22919.595,E2 22919.595} C_VEL
LIN {X 0,Y 513.852,Z 873.379,A -85,B 0,C 180,E1 22917.918,E2 22917.918} C_VEL
LIN {X 0,Y 515.614,Z 853.592,A -85,B 0,C 180,E1 22916.389,E2 22916.389} C_VEL
LIN {X 0,Y 517.226,Z 833.899,A -85,B 0,C 180,E1 22915.102,E2 22915.102} C_VEL
LIN {X 0,Y 518.954,Z 811.631,A -85,B 0,C 180,E1 22913.88,E2 22913.88} C_VEL
LIN {X 0,Y 520.292,Z 791.097,A -85,B 0,C 180,E1 22912.96,E2 22912.96} C_VEL
LIN {X 0,Y 521.624,Z 767.185,A -85,B 0,C 180,E1 22912.119,E2 22912.119} C_VEL
LIN {X 0,Y 522.526,Z 746.63,A -85,B 0,C 180,E1 22911.582,E2 22911.582} C_VEL
LIN {X 0,Y 523.263,Z 715.28,A -85,B 0,C 180,E1 22911.024,E2 22911.024} C_VEL
LIN {X 0,Y 526.659,Z 504.774,A -85,B 0,C 180,E1 22907.633,E2 22907.633} C_VEL
LIN {X 0,Y 528.066,Z 413.605,A -85,B 0,C 180,E1 22906.117,E2 22906.117} C_VEL
LIN {X 0,Y 526.806,Z 408.028,A -85,B 0,C 180,E1 22905.881,E2 22905.881} C_VEL
LIN {X 0,Y 514.848,Z 389.549,A -85,B 0,C 180,E1 22904.202,E2 22904.202} C_VEL
LIN {X 0,Y 507.964,Z 375.562,A -85,B 0,C 180,E1 22902.16,E2 22902.16} C_VEL
LIN {X 0,Y 506.09,Z 371.882,A -85,B 0,C 180,E1 22901.591,E2 22901.591} C_VEL
LIN {X 0,Y 504.674,Z 368.414,A -85,B 0,C 180,E1 22901.022,E2 22901.022} C_VEL
LIN {X 0,Y 504.695,Z 368.171,A -85,B 0,C 180,E1 22898.149,E2 22898.149} C_VEL
LIN {X 0,Y 504.634,Z 368.159,A -85,B 0,C 180,E1 22894.794,E2 22894.794} C_VEL
LIN {X 0,Y 504.629,Z 368.166,A -85,B 0,C 180,E1 22891.273,E2 22891.273} C_VEL
LIN {X 0,Y 504.701,Z 368.181,A -85,B 0,C 180,E1 22887.936,E2 22887.936} C_VEL
LIN {X 0,Y 504.628,Z 368.188,A -85,B 0,C 180,E1 22884.584,E2 22884.584} C_VEL
LIN {X 0,Y 504.633,Z 368.183,A -85,B 0,C 180,E1 22881.015,E2 22881.015} C_VEL
LIN {X 0,Y 504.692,Z 368.178,A -85,B 0,C 180,E1 22877.644,E2 22877.644} C_VEL
LIN {X 0,Y 504.633,Z 368.18,A -85,B 0,C 180,E1 22874.339,E2 22874.339} C_VEL
LIN {X 0,Y 504.646,Z 368.184,A -85,B 0,C 180,E1 22870.849,E2 22870.849} C_VEL
LIN {X 0,Y 504.688,Z 368.18,A -85,B 0,C 180,E1 22867.513,E2 22867.513} C_VEL
LIN {X 0,Y 504.639,Z 368.184,A -85,B 0,C 180,E1 22864.09,E2 22864.09} C_VEL
LIN {X 0,Y 504.656,Z 368.183,A -85,B 0,C 180,E1 22860.567,E2 22860.567} C_VEL
LIN {X 0,Y 504.687,Z 368.183,A -85,B 0,C 180,E1 22857.274,E2 22857.274} C_VEL
LIN {X 0,Y 504.646,Z 368.184,A -85,B 0,C 180,E1 22853.858,E2 22853.858} C_VEL
LIN {X 0,Y 504.677,Z 368.181,A -85,B 0,C 180,E1 22850.42,E2 22850.42} C_VEL
LIN {X 0,Y 504.686,Z 368.182,A -85,B 0,C 180,E1 22847.063,E2 22847.063} C_VEL
LIN {X 0,Y 504.653,Z 368.182,A -85,B 0,C 180,E1 22843.659,E2 22843.659} C_VEL
LIN {X 0,Y 504.691,Z 368.18,A -85,B 0,C 180,E1 22840.197,E2 22840.197} C_VEL
LIN {X 0,Y 504.69,Z 368.182,A -85,B 0,C 180,E1 22836.781,E2 22836.781} C_VEL
LIN {X 0,Y 504.661,Z 368.181,A -85,B 0,C 180,E1 22833.31,E2 22833.31} C_VEL
LIN {X 0,Y 504.7,Z 368.178,A -85,B 0,C 180,E1 22829.919,E2 22829.919} C_VEL
LIN {X 0,Y 504.699,Z 368.184,A -85,B 0,C 180,E1 22826.445,E2 22826.445} C_VEL
LIN {X 0,Y 504.667,Z 368.182,A -85,B 0,C 180,E1 22822.965,E2 22822.965} C_VEL
LIN {X 0,Y 504.693,Z 368.174,A -85,B 0,C 180,E1 22819.472,E2 22819.472} C_VEL
LIN {X 0,Y 504.709,Z 368.175,A -85,B 0,C 180,E1 22815.944,E2 22815.944} C_VEL
LIN {X 0,Y 504.676,Z 368.176,A -85,B 0,C 180,E1 22812.493,E2 22812.493} C_VEL
LIN {X 0,Y 504.699,Z 368.177,A -85,B 0,C 180,E1 22810.054,E2 22810.054} C_VEL
LIN {X 0,Y 503.731,Z 368.302,A -85,B 0,C 180,E1 22809.179,E2 22809.179} C_VEL
LIN {X 0,Y 497.265,Z 369.111,A -85,B 0,C 180,E1 22806.721,E2 22806.721} C_VEL
LIN {X 0,Y 496.753,Z 369.172,A -85,B 0,C 180,E1 22806.08,E2 22806.08} C_VEL
LIN {X 0,Y 496.74,Z 369.163,A -85,B 0,C 180,E1 22802.5,E2 22802.5} C_VEL
LIN {X 0,Y 496.766,Z 369.144,A -85,B 0,C 180,E1 22799.012,E2 22799.012} C_VEL
LIN {X 0,Y 496.766,Z 369.147,A -85,B 0,C 180,E1 22795.509,E2 22795.509} C_VEL
LIN {X 0,Y 496.744,Z 369.154,A -85,B 0,C 180,E1 22791.982,E2 22791.982} C_VEL
LIN {X 0,Y 496.764,Z 369.284,A -85,B 0,C 180,E1 22789.955,E2 22789.955} C_VEL
LIN {X 0,Y 497.118,Z 370.749,A -85,B 0,C 180,E1 22789.707,E2 22789.707} C_VEL
LIN {X 0,Y 499.09,Z 373.88,A -85,B 0,C 180,E1 22789.386,E2 22789.386} C_VEL
LIN {X 0,Y 500.711,Z 375.549,A -85,B 0,C 180,E1 22789.149,E2 22789.149} C_VEL
LIN {X 0,Y 503.45,Z 379.533,A -85,B 0,C 180,E1 22788.729,E2 22788.729} C_VEL
LIN {X 0,Y 512.332,Z 391.907,A -85,B 0,C 180,E1 22787.429,E2 22787.429} C_VEL
LIN {X 0,Y 522.132,Z 406.185,A -85,B 0,C 180,E1 22786.067,E2 22786.067} C_VEL
LIN {X 0,Y 518.078,Z 624.715,A -85,B 0,C 180,E1 22782.467,E2 22782.467} C_VEL
LIN {X 0,Y 516.467,Z 711.379,A -85,B 0,C 180,E1 22781.042,E2 22781.042} C_VEL
LIN {X 0,Y 515.492,Z 734.051,A -85,B 0,C 180,E1 22780.484,E2 22780.484} C_VEL
LIN {X 0,Y 514.161,Z 756.616,A -85,B 0,C 180,E1 22779.722,E2 22779.722} C_VEL
LIN {X 0,Y 512.583,Z 778.901,A -85,B 0,C 180,E1 22778.748,E2 22778.748} C_VEL
LIN {X 0,Y 510.858,Z 800.427,A -85,B 0,C 180,E1 22777.588,E2 22777.588} C_VEL
LIN {X 0,Y 509.003,Z 821.123,A -85,B 0,C 180,E1 22776.255,E2 22776.255} C_VEL
LIN {X 0,Y 507.001,Z 842.269,A -85,B 0,C 180,E1 22774.634,E2 22774.634} C_VEL
LIN {X 0,Y 505.044,Z 861.645,A -85,B 0,C 180,E1 22772.89,E2 22772.89} C_VEL
LIN {X 0,Y 503.263,Z 879.541,A -85,B 0,C 180,E1 22771.021,E2 22771.021} C_VEL
LIN {X 0,Y 501.485,Z 897.558,A -85,B 0,C 180,E1 22768.854,E2 22768.854} C_VEL
LIN {X 0,Y 500.042,Z 913.276,A -85,B 0,C 180,E1 22766.672,E2 22766.672} C_VEL
LIN {X 0,Y 498.812,Z 927.695,A -85,B 0,C 180,E1 22764.36,E2 22764.36} C_VEL
LIN {X 0,Y 497.774,Z 941.447,A -85,B 0,C 180,E1 22761.798,E2 22761.798} C_VEL
LIN {X 0,Y 497.013,Z 953.174,A -85,B 0,C 180,E1 22759.214,E2 22759.214} C_VEL
LIN {X 0,Y 496.499,Z 963.198,A -85,B 0,C 180,E1 22756.577,E2 22756.577} C_VEL
LIN {X 0,Y 496.188,Z 971.346,A -85,B 0,C 180,E1 22753.987,E2 22753.987} C_VEL
LIN {X 0,Y 496.024,Z 977.904,A -85,B 0,C 180,E1 22751.336,E2 22751.336} C_VEL
LIN {X 0,Y 495.937,Z 982.85,A -85,B 0,C 180,E1 22748.661,E2 22748.661} C_VEL
LIN {X 0,Y 495.905,Z 986.129,A -85,B 0,C 180,E1 22745.963,E2 22745.963} C_VEL
LIN {X 0,Y 495.906,Z 987.763,A -85,B 0,C 180,E1 22743.278,E2 22743.278} C_VEL
LIN {X 0,Y 495.918,Z 987.795,A -85,B 0,C 180,E1 22740.794,E2 22740.794} C_VEL
LIN {X 0,Y 495.911,Z 986.252,A -85,B 0,C 180,E1 22738.085,E2 22738.085} C_VEL
LIN {X 0,Y 495.929,Z 983.225,A -85,B 0,C 180,E1 22735.488,E2 22735.488} C_VEL
LIN {X 0,Y 496.011,Z 978.34,A -85,B 0,C 180,E1 22732.773,E2 22732.773} C_VEL
LIN {X 0,Y 496.166,Z 972.345,A -85,B 0,C 180,E1 22730.294,E2 22730.294} C_VEL
LIN {X 0,Y 496.466,Z 964.008,A -85,B 0,C 180,E1 22727.569,E2 22727.569} C_VEL
LIN {X 0,Y 496.94,Z 954.753,A -85,B 0,C 180,E1 22725.069,E2 22725.069} C_VEL
LIN {X 0,Y 497.66,Z 943.124,A -85,B 0,C 180,E1 22722.46,E2 22722.46} C_VEL
LIN {X 0,Y 498.651,Z 929.788,A -85,B 0,C 180,E1 22719.915,E2 22719.915} C_VEL
LIN {X 0,Y 499.879,Z 915.029,A -85,B 0,C 180,E1 22717.506,E2 22717.506} C_VEL
LIN {X 0,Y 501.392,Z 898.602,A -85,B 0,C 180,E1 22715.192,E2 22715.192} C_VEL
LIN {X 0,Y 503.12,Z 881.085,A -85,B 0,C 180,E1 22713.061,E2 22713.061} C_VEL
LIN {X 0,Y 504.949,Z 862.697,A -85,B 0,C 180,E1 22711.119,E2 22711.119} C_VEL
LIN {X 0,Y 506.934,Z 842.907,A -85,B 0,C 180,E1 22709.33,E2 22709.33} C_VEL
LIN {X 0,Y 508.859,Z 822.505,A -85,B 0,C 180,E1 22707.755,E2 22707.755} C_VEL
LIN {X 0,Y 510.771,Z 801.449,A -85,B 0,C 180,E1 22706.383,E2 22706.383} C_VEL
LIN {X 0,Y 512.489,Z 780.375,A -85,B 0,C 180,E1 22705.233,E2 22705.233} C_VEL
LIN {X 0,Y 514.097,Z 757.712,A -85,B 0,C 180,E1 22704.229,E2 22704.229} C_VEL
LIN {X 0,Y 515.435,Z 734.943,A -85,B 0,C 180,E1 22703.453,E2 22703.453} C_VEL
LIN {X 0,Y 516.414,Z 712.697,A -85,B 0,C 180,E1 22702.896,E2 22702.896} C_VEL
LIN {X 0,Y 517.345,Z 667.633,A -85,B 0,C 180,E1 22702.137,E2 22702.137} C_VEL
LIN {X 0,Y 521.149,Z 457.427,A -85,B 0,C 180,E1 22698.697,E2 22698.697} C_VEL
LIN {X 0,Y 522.03,Z 405.932,A -85,B 0,C 180,E1 22697.82,E2 22697.82} C_VEL
LIN {X 0,Y 510.672,Z 389.477,A -85,B 0,C 180,E1 22696.23,E2 22696.23} C_VEL
LIN {X 0,Y 503.537,Z 379.61,A -85,B 0,C 180,E1 22695.163,E2 22695.163} C_VEL
LIN {X 0,Y 500.777,Z 375.667,A -85,B 0,C 180,E1 22694.734,E2 22694.734} C_VEL
LIN {X 0,Y 499.721,Z 374.429,A -85,B 0,C 180,E1 22694.573,E2 22694.573} C_VEL
LIN {X 0,Y 497.484,Z 371.592,A -85,B 0,C 180,E1 22694.224,E2 22694.224} C_VEL
LIN {X 0,Y 496.937,Z 370.061,A -85,B 0,C 180,E1 22694.091,E2 22694.091} C_VEL
LIN {X 0,Y 496.77,Z 369.196,A -85,B 0,C 180,E1 22693.799,E2 22693.799} C_VEL
LIN {X 0,Y 496.766,Z 369.167,A -85,B 0,C 180,E1 22690.183,E2 22690.183} C_VEL
LIN {X 0,Y 496.754,Z 369.168,A -85,B 0,C 180,E1 22686.705,E2 22686.705} C_VEL
LIN {X 0,Y 496.764,Z 369.165,A -85,B 0,C 180,E1 22683.116,E2 22683.116} C_VEL
LIN {X 0,Y 496.75,Z 369.167,A -85,B 0,C 180,E1 22679.539,E2 22679.539} C_VEL
LIN {X 0,Y 496.761,Z 369.172,A -85,B 0,C 180,E1 22675.961,E2 22675.961} C_VEL
LIN {X 0,Y 496.769,Z 369.17,A -85,B 0,C 180,E1 22672.367,E2 22672.367} C_VEL
LIN {X 0,Y 496.752,Z 369.167,A -85,B 0,C 180,E1 22668.859,E2 22668.859} C_VEL
LIN {X 0,Y 496.733,Z 369.172,A -85,B 0,C 180,E1 22665.309,E2 22665.309} C_VEL
LIN {X 0,Y 496.761,Z 369.171,A -85,B 0,C 180,E1 22661.813,E2 22661.813} C_VEL
LIN {X 0,Y 496.767,Z 369.165,A -85,B 0,C 180,E1 22658.264,E2 22658.264} C_VEL
LIN {X 0,Y 496.717,Z 369.174,A -85,B 0,C 180,E1 22654.867,E2 22654.867} C_VEL
LIN {X 0,Y 496.726,Z 369.168,A -85,B 0,C 180,E1 22651.36,E2 22651.36} C_VEL
LIN {X 0,Y 496.761,Z 369.164,A -85,B 0,C 180,E1 22647.93,E2 22647.93} C_VEL
LIN {X 0,Y 496.699,Z 369.178,A -85,B 0,C 180,E1 22644.568,E2 22644.568} C_VEL
LIN {X 0,Y 496.692,Z 369.174,A -85,B 0,C 180,E1 22640.945,E2 22640.945} C_VEL
LIN {X 0,Y 496.784,Z 369.454,A -85,B 0,C 180,E1 22639.796,E2 22639.796} C_VEL
LIN {X 0,Y 498.423,Z 373.231,A -85,B 0,C 180,E1 22639.159,E2 22639.159} C_VEL
LIN {X 0,Y 503.937,Z 384.485,A -85,B 0,C 180,E1 22637.424,E2 22637.424} C_VEL
LIN {X 0,Y 506.331,Z 389.138,A -85,B 0,C 180,E1 22636.773,E2 22636.773} C_VEL
LIN {X 0,Y 521.685,Z 412.757,A -85,B 0,C 180,E1 22634.562,E2 22634.562} C_VEL
LIN {X 0,Y 522.328,Z 417.339,A -85,B 0,C 180,E1 22634.407,E2 22634.407} C_VEL
LIN {X 0,Y 518.509,Z 625.8,A -85,B 0,C 180,E1 22630.972,E2 22630.972} C_VEL
LIN {X 0,Y 516.495,Z 739.954,A -85,B 0,C 180,E1 22629.113,E2 22629.113} C_VEL
LIN {X 0,Y 515.508,Z 763.015,A -85,B 0,C 180,E1 22628.553,E2 22628.553} C_VEL
LIN {X 0,Y 514.401,Z 782.775,A -85,B 0,C 180,E1 22627.907,E2 22627.907} C_VEL
LIN {X 0,Y 512.762,Z 806.22,A -85,B 0,C 180,E1 22626.92,E2 22626.92} C_VEL
LIN {X 0,Y 511.111,Z 827.661,A -85,B 0,C 180,E1 22625.8,E2 22625.8} C_VEL
LIN {X 0,Y 509.273,Z 848.096,A -85,B 0,C 180,E1 22624.503,E2 22624.503} C_VEL
LIN {X 0,Y 507.387,Z 868.15,A -85,B 0,C 180,E1 22623.019,E2 22623.019} C_VEL
LIN {X 0,Y 505.493,Z 887.237,A -85,B 0,C 180,E1 22621.349,E2 22621.349} C_VEL
LIN {X 0,Y 503.525,Z 906.762,A -85,B 0,C 180,E1 22619.374,E2 22619.374} C_VEL
LIN {X 0,Y 501.933,Z 923.13,A -85,B 0,C 180,E1 22617.464,E2 22617.464} C_VEL
LIN {X 0,Y 500.416,Z 939.123,A -85,B 0,C 180,E1 22615.317,E2 22615.317} C_VEL
LIN {X 0,Y 499.166,Z 953.49,A -85,B 0,C 180,E1 22613.119,E2 22613.119} C_VEL
LIN {X 0,Y 498.079,Z 967.072,A -85,B 0,C 180,E1 22610.693,E2 22610.693} C_VEL
LIN {X 0,Y 497.254,Z 979.275,A -85,B 0,C 180,E1 22608.163,E2 22608.163} C_VEL
LIN {X 0,Y 496.697,Z 989.057,A -85,B 0,C 180,E1 22605.772,E2 22605.772} C_VEL
LIN {X 0,Y 496.295,Z 998.338,A -85,B 0,C 180,E1 22603.044,E2 22603.044} C_VEL
LIN {X 0,Y 496.085,Z 1004.858,A -85,B 0,C 180,E1 22600.689,E2 22600.689} C_VEL
LIN {X 0,Y 495.974,Z 1010.629,A -85,B 0,C 180,E1 22597.999,E2 22597.999} C_VEL
LIN {X 0,Y 495.911,Z 1014.432,A -85,B 0,C 180,E1 22595.557,E2 22595.557} C_VEL
LIN {X 0,Y 495.892,Z 1016.984,A -85,B 0,C 180,E1 22592.893,E2 22592.893} C_VEL
LIN {X 0,Y 495.884,Z 1017.894,A -85,B 0,C 180,E1 22590.581,E2 22590.581} C_VEL
LIN {X 0,Y 495.914,Z 1017.394,A -85,B 0,C 180,E1 22587.808,E2 22587.808} C_VEL
LIN {X 0,Y 495.906,Z 1015.505,A -85,B 0,C 180,E1 22585.378,E2 22585.378} C_VEL
LIN {X 0,Y 495.924,Z 1011.881,A -85,B 0,C 180,E1 22582.707,E2 22582.707} C_VEL
LIN {X 0,Y 496.008,Z 1007.327,A -85,B 0,C 180,E1 22580.372,E2 22580.372} C_VEL
LIN {X 0,Y 496.208,Z 1000.743,A -85,B 0,C 180,E1 22577.76,E2 22577.76} C_VEL
LIN {X 0,Y 496.518,Z 992.951,A -85,B 0,C 180,E1 22575.306,E2 22575.306} C_VEL
LIN {X 0,Y 497.063,Z 982.41,A -85,B 0,C 180,E1 22572.564,E2 22572.564} C_VEL
LIN {X 0,Y 497.777,Z 971.436,A -85,B 0,C 180,E1 22570.16,E2 22570.16} C_VEL
LIN {X 0,Y 498.75,Z 958.48,A -85,B 0,C 180,E1 22567.74,E2 22567.74} C_VEL
LIN {X 0,Y 499.969,Z 944.245,A -85,B 0,C 180,E1 22565.425,E2 22565.425} C_VEL
LIN {X 0,Y 501.403,Z 928.445,A -85,B 0,C 180,E1 22563.218,E2 22563.218} C_VEL
LIN {X 0,Y 503.197,Z 910.159,A -85,B 0,C 180,E1 22561.004,E2 22561.004} C_VEL
LIN {X 0,Y 505.032,Z 891.955,A -85,B 0,C 180,E1 22559.091,E2 22559.091} C_VEL
LIN {X 0,Y 506.916,Z 872.826,A -85,B 0,C 180,E1 22557.375,E2 22557.375} C_VEL
LIN {X 0,Y 508.848,Z 852.705,A -85,B 0,C 180,E1 22555.813,E2 22555.813} C_VEL
LIN {X 0,Y 510.623,Z 832.991,A -85,B 0,C 180,E1 22554.521,E2 22554.521} C_VEL
LIN {X 0,Y 512.467,Z 810.472,A -85,B 0,C 180,E1 22553.286,E2 22553.286} C_VEL
LIN {X 0,Y 513.939,Z 789.615,A -85,B 0,C 180,E1 22552.353,E2 22552.353} C_VEL
LIN {X 0,Y 515.316,Z 766.662,A -85,B 0,C 180,E1 22551.554,E2 22551.554} C_VEL
LIN {X 0,Y 516.264,Z 746.467,A -85,B 0,C 180,E1 22551.025,E2 22551.025} C_VEL
LIN {X 0,Y 517.039,Z 715.438,A -85,B 0,C 180,E1 22550.468,E2 22550.468} C_VEL
LIN {X 0,Y 520.686,Z 506.52,A -85,B 0,C 180,E1 22547.07,E2 22547.07} C_VEL
LIN {X 0,Y 522.241,Z 415.425,A -85,B 0,C 180,E1 22545.539,E2 22545.539} C_VEL
LIN {X 0,Y 521.413,Z 412.278,A -85,B 0,C 180,E1 22545.39,E2 22545.39} C_VEL
LIN {X 0,Y 506.262,Z 389.027,A -85,B 0,C 180,E1 22543.182,E2 22543.182} C_VEL
LIN {X 0,Y 500.427,Z 377.299,A -85,B 0,C 180,E1 22541.402,E2 22541.402} C_VEL
LIN {X 0,Y 496.837,Z 369.662,A -85,B 0,C 180,E1 22540.176,E2 22540.176} C_VEL
LIN {X 0,Y 496.698,Z 369.143,A -85,B 0,C 180,E1 22539.566,E2 22539.566} C_VEL
LIN {X 0,Y 496.752,Z 369.144,A -85,B 0,C 180,E1 22536.193,E2 22536.193} C_VEL
LIN {X 0,Y 496.699,Z 369.178,A -85,B 0,C 180,E1 22532.718,E2 22532.718} C_VEL
LIN {X 0,Y 496.687,Z 369.16,A -85,B 0,C 180,E1 22529.154,E2 22529.154} C_VEL
LIN {X 0,Y 496.748,Z 369.166,A -85,B 0,C 180,E1 22525.891,E2 22525.891} C_VEL
LIN {X 0,Y 496.69,Z 369.173,A -85,B 0,C 180,E1 22522.487,E2 22522.487} C_VEL
LIN {X 0,Y 496.694,Z 369.175,A -85,B 0,C 180,E1 22518.91,E2 22518.91} C_VEL
LIN {X 0,Y 496.761,Z 369.167,A -85,B 0,C 180,E1 22515.527,E2 22515.527} C_VEL
LIN {X 0,Y 496.699,Z 369.173,A -85,B 0,C 180,E1 22512.202,E2 22512.202} C_VEL
LIN {X 0,Y 496.699,Z 369.167,A -85,B 0,C 180,E1 22508.566,E2 22508.566} C_VEL
LIN {X 0,Y 496.759,Z 369.165,A -85,B 0,C 180,E1 22505.196,E2 22505.196} C_VEL
LIN {X 0,Y 496.716,Z 369.167,A -85,B 0,C 180,E1 22501.73,E2 22501.73} C_VEL
LIN {X 0,Y 496.707,Z 369.17,A -85,B 0,C 180,E1 22498.269,E2 22498.269} C_VEL
LIN {X 0,Y 496.759,Z 369.168,A -85,B 0,C 180,E1 22494.803,E2 22494.803} C_VEL
LIN {X 0,Y 496.723,Z 369.166,A -85,B 0,C 180,E1 22491.433,E2 22491.433} C_VEL
LIN {X 0,Y 496.713,Z 369.169,A -85,B 0,C 180,E1 22487.915,E2 22487.915} C_VEL
LIN {X 0,Y 496.765,Z 369.168,A -85,B 0,C 180,E1 22484.472,E2 22484.472} C_VEL
LIN {X 0,Y 496.742,Z 369.166,A -85,B 0,C 180,E1 22480.969,E2 22480.969} C_VEL
LIN {X 0,Y 496.719,Z 369.168,A -85,B 0,C 180,E1 22477.493,E2 22477.493} C_VEL
LIN {X 0,Y 496.762,Z 369.168,A -85,B 0,C 180,E1 22474.102,E2 22474.102} C_VEL
LIN {X 0,Y 496.751,Z 369.167,A -85,B 0,C 180,E1 22470.627,E2 22470.627} C_VEL
LIN {X 0,Y 496.725,Z 369.169,A -85,B 0,C 180,E1 22467.216,E2 22467.216} C_VEL
LIN {X 0,Y 496.759,Z 369.168,A -85,B 0,C 180,E1 22463.718,E2 22463.718} C_VEL
LIN {X 0,Y 496.771,Z 369.17,A -85,B 0,C 180,E1 22460.204,E2 22460.204} C_VEL
LIN {X 0,Y 496.735,Z 369.171,A -85,B 0,C 180,E1 22456.655,E2 22456.655} C_VEL
LIN {X 0,Y 496.738,Z 369.162,A -85,B 0,C 180,E1 22453.021,E2 22453.021} C_VEL
LIN {X 0,Y 496.771,Z 369.168,A -85,B 0,C 180,E1 22449.567,E2 22449.567} C_VEL
LIN {X 0,Y 496.753,Z 369.172,A -85,B 0,C 180,E1 22446.08,E2 22446.08} C_VEL
LIN {X 0,Y 495.786,Z 369.287,A -85,B 0,C 180,E1 22445.191,E2 22445.191} C_VEL
LIN {X 0,Y 489.325,Z 370.084,A -85,B 0,C 180,E1 22442.693,E2 22442.693} C_VEL
LIN {X 0,Y 488.811,Z 370.155,A -85,B 0,C 180,E1 22442.041,E2 22442.041} C_VEL
LIN {X 0,Y 488.803,Z 370.139,A -85,B 0,C 180,E1 22438.408,E2 22438.408} C_VEL
LIN {X 0,Y 488.825,Z 370.132,A -85,B 0,C 180,E1 22434.915,E2 22434.915} C_VEL
LIN {X 0,Y 488.828,Z 370.132,A -85,B 0,C 180,E1 22431.347,E2 22431.347} C_VEL
LIN {X 0,Y 488.842,Z 370.264,A -85,B 0,C 180,E1 22430.969,E2 22430.969} C_VEL
LIN {X 0,Y 489.189,Z 371.711,A -85,B 0,C 180,E1 22430.719,E2 22430.719} C_VEL
LIN {X 0,Y 491.057,Z 374.769,A -85,B 0,C 180,E1 22430.397,E2 22430.397} C_VEL
LIN {X 0,Y 492.796,Z 376.508,A -85,B 0,C 180,E1 22430.132,E2 22430.132} C_VEL
LIN {X 0,Y 495.451,Z 380.451,A -85,B 0,C 180,E1 22429.705,E2 22429.705} C_VEL
LIN {X 0,Y 497.071,Z 382.51,A -85,B 0,C 180,E1 22429.456,E2 22429.456} C_VEL
LIN {X 0,Y 507.849,Z 397.455,A -85,B 0,C 180,E1 22427.838,E2 22427.838} C_VEL
LIN {X 0,Y 516.331,Z 409.996,A -85,B 0,C 180,E1 22426.625,E2 22426.625} C_VEL
LIN {X 0,Y 511.928,Z 627.816,A -85,B 0,C 180,E1 22422.997,E2 22422.997} C_VEL
LIN {X 0,Y 510.226,Z 711.917,A -85,B 0,C 180,E1 22421.598,E2 22421.598} C_VEL
LIN {X 0,Y 509.169,Z 734.742,A -85,B 0,C 180,E1 22421.027,E2 22421.027} C_VEL
LIN {X 0,Y 507.761,Z 757.15,A -85,B 0,C 180,E1 22420.262,E2 22420.262} C_VEL
LIN {X 0,Y 506.032,Z 779.652,A -85,B 0,C 180,E1 22419.263,E2 22419.263} C_VEL
LIN {X 0,Y 504.17,Z 801.066,A -85,B 0,C 180,E1 22418.091,E2 22418.091} C_VEL
LIN {X 0,Y 502.173,Z 821.68,A -85,B 0,C 180,E1 22416.743,E2 22416.743} C_VEL
LIN {X 0,Y 500.072,Z 842.13,A -85,B 0,C 180,E1 22415.158,E2 22415.158} C_VEL
LIN {X 0,Y 497.965,Z 861.521,A -85,B 0,C 180,E1 22413.392,E2 22413.392} C_VEL
LIN {X 0,Y 496.005,Z 879.458,A -85,B 0,C 180,E1 22411.498,E2 22411.498} C_VEL
LIN {X 0,Y 494.068,Z 897.488,A -85,B 0,C 180,E1 22409.301,E2 22409.301} C_VEL
LIN {X 0,Y 492.489,Z 913.212,A -85,B 0,C 180,E1 22407.087,E2 22407.087} C_VEL
LIN {X 0,Y 491.081,Z 928.211,A -85,B 0,C 180,E1 22404.641,E2 22404.641} C_VEL
LIN {X 0,Y 489.933,Z 941.963,A -85,B 0,C 180,E1 22402.02,E2 22402.02} C_VEL
LIN {X 0,Y 489.131,Z 953.188,A -85,B 0,C 180,E1 22399.497,E2 22399.497} C_VEL
LIN {X 0,Y 488.57,Z 963.04,A -85,B 0,C 180,E1 22396.867,E2 22396.867} C_VEL
LIN {X 0,Y 488.22,Z 971.123,A -85,B 0,C 180,E1 22394.271,E2 22394.271} C_VEL
LIN {X 0,Y 488.037,Z 977.791,A -85,B 0,C 180,E1 22391.545,E2 22391.545} C_VEL
LIN {X 0,Y 487.937,Z 982.79,A -85,B 0,C 180,E1 22388.808,E2 22388.808} C_VEL
LIN {X 0,Y 487.895,Z 985.989,A -85,B 0,C 180,E1 22386.186,E2 22386.186} C_VEL
LIN {X 0,Y 487.89,Z 987.707,A -85,B 0,C 180,E1 22383.582,E2 22383.582} C_VEL
LIN {X 0,Y 487.913,Z 987.848,A -85,B 0,C 180,E1 22381.05,E2 22381.05} C_VEL
LIN {X 0,Y 487.909,Z 986.459,A -85,B 0,C 180,E1 22378.261,E2 22378.261} C_VEL
LIN {X 0,Y 487.919,Z 983.622,A -85,B 0,C 180,E1 22375.674,E2 22375.674} C_VEL
LIN {X 0,Y 487.988,Z 979.192,A -85,B 0,C 180,E1 22373.044,E2 22373.044} C_VEL
LIN {X 0,Y 488.169,Z 973.042,A -85,B 0,C 180,E1 22370.365,E2 22370.365} C_VEL
LIN {X 0,Y 488.488,Z 965.058,A -85,B 0,C 180,E1 22367.639,E2 22367.639} C_VEL
LIN {X 0,Y 488.996,Z 955.686,A -85,B 0,C 180,E1 22365.03,E2 22365.03} C_VEL
LIN {X 0,Y 489.781,Z 944.142,A -85,B 0,C 180,E1 22362.351,E2 22362.351} C_VEL
LIN {X 0,Y 490.813,Z 931.27,A -85,B 0,C 180,E1 22359.822,E2 22359.822} C_VEL
LIN {X 0,Y 492.144,Z 916.659,A -85,B 0,C 180,E1 22357.357,E2 22357.357} C_VEL
LIN {X 0,Y 493.745,Z 900.798,A -85,B 0,C 180,E1 22355.048,E2 22355.048} C_VEL
LIN {X 0,Y 495.601,Z 883.494,A -85,B 0,C 180,E1 22352.868,E2 22352.868} C_VEL
LIN {X 0,Y 497.543,Z 865.309,A -85,B 0,C 180,E1 22350.894,E2 22350.894} C_VEL
LIN {X 0,Y 499.632,Z 846.098,A -85,B 0,C 180,E1 22349.097,E2 22349.097} C_VEL
LIN {X 0,Y 501.724,Z 825.964,A -85,B 0,C 180,E1 22347.481,E2 22347.481} C_VEL
LIN {X 0,Y 503.774,Z 805.406,A -85,B 0,C 180,E1 22346.08,E2 22346.08} C_VEL
LIN {X 0,Y 505.623,Z 784.868,A -85,B 0,C 180,E1 22344.911,E2 22344.911} C_VEL
LIN {X 0,Y 507.357,Z 762.731,A -85,B 0,C 180,E1 22343.874,E2 22343.874} C_VEL
LIN {X 0,Y 508.929,Z 738.486,A -85,B 0,C 180,E1 22342.998,E2 22342.998} C_VEL
LIN {X 0,Y 510.061,Z 715.791,A -85,B 0,C 180,E1 22342.398,E2 22342.398} C_VEL
LIN {X 0,Y 510.917,Z 681.821,A -85,B 0,C 180,E1 22341.795,E2 22341.795} C_VEL
LIN {X 0,Y 514.999,Z 473.024,A -85,B 0,C 180,E1 22338.347,E2 22338.347} C_VEL
LIN {X 0,Y 516.245,Z 409.517,A -85,B 0,C 180,E1 22337.257,E2 22337.257} C_VEL
LIN {X 0,Y 503.17,Z 390.783,A -85,B 0,C 180,E1 22335.355,E2 22335.355} C_VEL
LIN {X 0,Y 498.836,Z 384.995,A -85,B 0,C 180,E1 22334.688,E2 22334.688} C_VEL
LIN {X 0,Y 495.843,Z 380.803,A -85,B 0,C 180,E1 22334.212,E2 22334.212} C_VEL
LIN {X 0,Y 493.091,Z 376.989,A -85,B 0,C 180,E1 22333.766,E2 22333.766} C_VEL
LIN {X 0,Y 492.093,Z 375.642,A -85,B 0,C 180,E1 22333.603,E2 22333.603} C_VEL
LIN {X 0,Y 489.706,Z 372.937,A -85,B 0,C 180,E1 22333.22,E2 22333.22} C_VEL
LIN {X 0,Y 488.93,Z 370.855,A -85,B 0,C 180,E1 22333,E2 22333} C_VEL
LIN {X 0,Y 488.811,Z 370.166,A -85,B 0,C 180,E1 22332.643,E2 22332.643} C_VEL
LIN {X 0,Y 488.82,Z 370.156,A -85,B 0,C 180,E1 22329.062,E2 22329.062} C_VEL
LIN {X 0,Y 488.82,Z 370.152,A -85,B 0,C 180,E1 22325.517,E2 22325.517} C_VEL
LIN {X 0,Y 488.821,Z 370.157,A -85,B 0,C 180,E1 22321.876,E2 22321.876} C_VEL
LIN {X 0,Y 488.825,Z 370.16,A -85,B 0,C 180,E1 22318.36,E2 22318.36} C_VEL
LIN {X 0,Y 488.828,Z 370.152,A -85,B 0,C 180,E1 22314.719,E2 22314.719} C_VEL
LIN {X 0,Y 488.805,Z 370.159,A -85,B 0,C 180,E1 22311.176,E2 22311.176} C_VEL
LIN {X 0,Y 488.805,Z 370.16,A -85,B 0,C 180,E1 22307.598,E2 22307.598} C_VEL
LIN {X 0,Y 488.831,Z 370.158,A -85,B 0,C 180,E1 22304.093,E2 22304.093} C_VEL
LIN {X 0,Y 488.813,Z 370.159,A -85,B 0,C 180,E1 22300.524,E2 22300.524} C_VEL
LIN {X 0,Y 488.781,Z 370.158,A -85,B 0,C 180,E1 22297.002,E2 22297.002} C_VEL
LIN {X 0,Y 488.798,Z 370.154,A -85,B 0,C 180,E1 22293.518,E2 22293.518} C_VEL
LIN {X 0,Y 488.82,Z 370.153,A -85,B 0,C 180,E1 22290.061,E2 22290.061} C_VEL
LIN {X 0,Y 488.766,Z 370.166,A -85,B 0,C 180,E1 22286.581,E2 22286.581} C_VEL
LIN {X 0,Y 488.758,Z 370.163,A -85,B 0,C 180,E1 22282.926,E2 22282.926} C_VEL
LIN {X 0,Y 488.786,Z 370.417,A -85,B 0,C 180,E1 22280.796,E2 22280.796} C_VEL
LIN {X 0,Y 490.242,Z 373.892,A -85,B 0,C 180,E1 22280.178,E2 22280.178} C_VEL
LIN {X 0,Y 491.357,Z 375.841,A -85,B 0,C 180,E1 22279.83,E2 22279.83} C_VEL
LIN {X 0,Y 497.635,Z 388.275,A -85,B 0,C 180,E1 22277.87,E2 22277.87} C_VEL
LIN {X 0,Y 511.426,Z 409.361,A -85,B 0,C 180,E1 22275.757,E2 22275.757} C_VEL
LIN {X 0,Y 516.52,Z 417.767,A -85,B 0,C 180,E1 22275.025,E2 22275.025} C_VEL
LIN {X 0,Y 512.735,Z 607.522,A -85,B 0,C 180,E1 22271.849,E2 22271.849} C_VEL
LIN {X 0,Y 510.199,Z 740.237,A -85,B 0,C 180,E1 22269.665,E2 22269.665} C_VEL
LIN {X 0,Y 509.159,Z 763.157,A -85,B 0,C 180,E1 22269.104,E2 22269.104} C_VEL
LIN {X 0,Y 507.978,Z 783.456,A -85,B 0,C 180,E1 22268.438,E2 22268.438} C_VEL
LIN {X 0,Y 506.392,Z 805.046,A -85,B 0,C 180,E1 22267.529,E2 22267.529} C_VEL
LIN {X 0,Y 504.635,Z 825.842,A -85,B 0,C 180,E1 22266.446,E2 22266.446} C_VEL
LIN {X 0,Y 502.617,Z 847.192,A -85,B 0,C 180,E1 22265.096,E2 22265.096} C_VEL
LIN {X 0,Y 500.647,Z 866.592,A -85,B 0,C 180,E1 22263.659,E2 22263.659} C_VEL
LIN {X 0,Y 498.562,Z 885.9,A -85,B 0,C 180,E1 22261.971,E2 22261.971} C_VEL
LIN {X 0,Y 496.551,Z 904.541,A -85,B 0,C 180,E1 22260.095,E2 22260.095} C_VEL
LIN {X 0,Y 494.753,Z 921.102,A -85,B 0,C 180,E1 22258.16,E2 22258.16} C_VEL
LIN {X 0,Y 492.961,Z 938.276,A -85,B 0,C 180,E1 22255.857,E2 22255.857} C_VEL
LIN {X 0,Y 491.519,Z 953.49,A -85,B 0,C 180,E1 22253.5,E2 22253.5} C_VEL
LIN {X 0,Y 490.322,Z 967.07,A -85,B 0,C 180,E1 22251.035,E2 22251.035} C_VEL
LIN {X 0,Y 489.405,Z 979.276,A -85,B 0,C 180,E1 22248.464,E2 22248.464} C_VEL
LIN {X 0,Y 488.785,Z 989.055,A -85,B 0,C 180,E1 22246.034,E2 22246.034} C_VEL
LIN {X 0,Y 488.338,Z 998.339,A -85,B 0,C 180,E1 22243.26,E2 22243.26} C_VEL
LIN {X 0,Y 488.1,Z 1004.857,A -85,B 0,C 180,E1 22240.866,E2 22240.866} C_VEL
LIN {X 0,Y 487.981,Z 1010.629,A -85,B 0,C 180,E1 22238.131,E2 22238.131} C_VEL
LIN {X 0,Y 487.912,Z 1014.433,A -85,B 0,C 180,E1 22235.648,E2 22235.648} C_VEL
LIN {X 0,Y 487.89,Z 1016.984,A -85,B 0,C 180,E1 22232.94,E2 22232.94} C_VEL
LIN {X 0,Y 487.885,Z 1017.894,A -85,B 0,C 180,E1 22230.591,E2 22230.591} C_VEL
LIN {X 0,Y 487.914,Z 1017.394,A -85,B 0,C 180,E1 22227.772,E2 22227.772} C_VEL
LIN {X 0,Y 487.906,Z 1015.505,A -85,B 0,C 180,E1 22225.302,E2 22225.302} C_VEL
LIN {X 0,Y 487.932,Z 1011.881,A -85,B 0,C 180,E1 22222.586,E2 22222.586} C_VEL
LIN {X 0,Y 488.017,Z 1007.347,A -85,B 0,C 180,E1 22220.222,E2 22220.222} C_VEL
LIN {X 0,Y 488.241,Z 1000.832,A -85,B 0,C 180,E1 22217.587,E2 22217.587} C_VEL
LIN {X 0,Y 488.593,Z 992.951,A -85,B 0,C 180,E1 22215.062,E2 22215.062} C_VEL
LIN {X 0,Y 489.198,Z 982.339,A -85,B 0,C 180,E1 22212.258,E2 22212.258} C_VEL
LIN {X 0,Y 489.978,Z 971.434,A -85,B 0,C 180,E1 22209.83,E2 22209.83} C_VEL
LIN {X 0,Y 491.057,Z 958.478,A -85,B 0,C 180,E1 22207.372,E2 22207.372} C_VEL
LIN {X 0,Y 492.403,Z 944.243,A -85,B 0,C 180,E1 22205.021,E2 22205.021} C_VEL
LIN {X 0,Y 493.961,Z 928.444,A -85,B 0,C 180,E1 22202.782,E2 22202.782} C_VEL
LIN {X 0,Y 495.924,Z 910.158,A -85,B 0,C 180,E1 22200.537,E2 22200.537} C_VEL
LIN {X 0,Y 497.857,Z 892.57,A -85,B 0,C 180,E1 22198.663,E2 22198.663} C_VEL
LIN {X 0,Y 499.909,Z 873.372,A -85,B 0,C 180,E1 22196.911,E2 22196.911} C_VEL
LIN {X 0,Y 501.985,Z 853.574,A -85,B 0,C 180,E1 22195.347,E2 22195.347} C_VEL
LIN {X 0,Y 503.894,Z 833.892,A -85,B 0,C 180,E1 22194.037,E2 22194.037} C_VEL
LIN {X 0,Y 505.798,Z 812.781,A -85,B 0,C 180,E1 22192.848,E2 22192.848} C_VEL
LIN {X 0,Y 507.329,Z 792.546,A -85,B 0,C 180,E1 22191.918,E2 22191.918} C_VEL
LIN {X 0,Y 508.844,Z 769.287,A -85,B 0,C 180,E1 22191.074,E2 22191.074} C_VEL
LIN {X 0,Y 509.87,Z 748.725,A -85,B 0,C 180,E1 22190.518,E2 22190.518} C_VEL
LIN {X 0,Y 510.711,Z 721.324,A -85,B 0,C 180,E1 22189.999,E2 22189.999} C_VEL
LIN {X 0,Y 514.634,Z 514.631,A -85,B 0,C 180,E1 22186.6,E2 22186.6} C_VEL
LIN {X 0,Y 516.477,Z 417.304,A -85,B 0,C 180,E1 22184.949,E2 22184.949} C_VEL
LIN {X 0,Y 501.537,Z 394.351,A -85,B 0,C 180,E1 22182.751,E2 22182.751} C_VEL
LIN {X 0,Y 497.769,Z 388.671,A -85,B 0,C 180,E1 22182.136,E2 22182.136} C_VEL
LIN {X 0,Y 490.872,Z 374.663,A -85,B 0,C 180,E1 22179.912,E2 22179.912} C_VEL
LIN {X 0,Y 489.033,Z 371.458,A -85,B 0,C 180,E1 22179.332,E2 22179.332} C_VEL
LIN {X 0,Y 488.779,Z 370.315,A -85,B 0,C 180,E1 22179.096,E2 22179.096} C_VEL
LIN {X 0,Y 488.771,Z 370.13,A -85,B 0,C 180,E1 22175.662,E2 22175.662} C_VEL
LIN {X 0,Y 488.809,Z 370.151,A -85,B 0,C 180,E1 22172.141,E2 22172.141} C_VEL
LIN {X 0,Y 488.75,Z 370.157,A -85,B 0,C 180,E1 22168.734,E2 22168.734} C_VEL
LIN {X 0,Y 488.756,Z 370.166,A -85,B 0,C 180,E1 22165.182,E2 22165.182} C_VEL
LIN {X 0,Y 488.82,Z 370.161,A -85,B 0,C 180,E1 22161.729,E2 22161.729} C_VEL
LIN {X 0,Y 488.764,Z 370.165,A -85,B 0,C 180,E1 22158.239,E2 22158.239} C_VEL
LIN {X 0,Y 488.753,Z 370.157,A -85,B 0,C 180,E1 22154.694,E2 22154.694} C_VEL
LIN {X 0,Y 488.811,Z 370.155,A -85,B 0,C 180,E1 22151.324,E2 22151.324} C_VEL
LIN {X 0,Y 488.774,Z 370.157,A -85,B 0,C 180,E1 22147.877,E2 22147.877} C_VEL
LIN {X 0,Y 488.762,Z 370.161,A -85,B 0,C 180,E1 22144.34,E2 22144.34} C_VEL
LIN {X 0,Y 488.814,Z 370.161,A -85,B 0,C 180,E1 22140.937,E2 22140.937} C_VEL
LIN {X 0,Y 488.785,Z 370.16,A -85,B 0,C 180,E1 22137.537,E2 22137.537} C_VEL
LIN {X 0,Y 488.768,Z 370.161,A -85,B 0,C 180,E1 22134.011,E2 22134.011} C_VEL
LIN {X 0,Y 488.814,Z 370.159,A -85,B 0,C 180,E1 22130.581,E2 22130.581} C_VEL
LIN {X 0,Y 488.803,Z 370.16,A -85,B 0,C 180,E1 22127.116,E2 22127.116} C_VEL
LIN {X 0,Y 488.776,Z 370.16,A -85,B 0,C 180,E1 22123.724,E2 22123.724} C_VEL
LIN {X 0,Y 488.819,Z 370.158,A -85,B 0,C 180,E1 22120.275,E2 22120.275} C_VEL
LIN {X 0,Y 488.816,Z 370.16,A -85,B 0,C 180,E1 22116.747,E2 22116.747} C_VEL
LIN {X 0,Y 488.784,Z 370.16,A -85,B 0,C 180,E1 22113.254,E2 22113.254} C_VEL
LIN {X 0,Y 488.811,Z 370.157,A -85,B 0,C 180,E1 22109.788,E2 22109.788} C_VEL
LIN {X 0,Y 488.826,Z 370.159,A -85,B 0,C 180,E1 22106.336,E2 22106.336} C_VEL
LIN {X 0,Y 488.792,Z 370.161,A -85,B 0,C 180,E1 22102.882,E2 22102.882} C_VEL
LIN {X 0,Y 488.8,Z 370.153,A -85,B 0,C 180,E1 22099.267,E2 22099.267} C_VEL
LIN {X 0,Y 488.831,Z 370.152,A -85,B 0,C 180,E1 22095.709,E2 22095.709} C_VEL
LIN {X 0,Y 488.818,Z 370.155,A -85,B 0,C 180,E1 22092.131,E2 22092.131} C_VEL
LIN {X 0,Y 488.798,Z 370.16,A -85,B 0,C 180,E1 22088.595,E2 22088.595} C_VEL
LIN {X 0,Y 488.822,Z 370.147,A -85,B 0,C 180,E1 22085.078,E2 22085.078} C_VEL
LIN {X 0,Y 488.811,Z 370.155,A -85,B 0,C 180,E1 22082.041,E2 22082.041} C_VEL
LIN {X 0,Y 487.844,Z 370.279,A -85,B 0,C 180,E1 22081.138,E2 22081.138} C_VEL
LIN {X 0,Y 481.386,Z 371.061,A -85,B 0,C 180,E1 22078.599,E2 22078.599} C_VEL
LIN {X 0,Y 480.872,Z 371.134,A -85,B 0,C 180,E1 22077.937,E2 22077.937} C_VEL
LIN {X 0,Y 480.866,Z 371.125,A -85,B 0,C 180,E1 22074.307,E2 22074.307} C_VEL
LIN {X 0,Y 480.887,Z 371.284,A -85,B 0,C 180,E1 22072.038,E2 22072.038} C_VEL
LIN {X 0,Y 481.238,Z 372.716,A -85,B 0,C 180,E1 22071.787,E2 22071.787} C_VEL
LIN {X 0,Y 483.139,Z 375.756,A -85,B 0,C 180,E1 22071.445,E2 22071.445} C_VEL
LIN {X 0,Y 484.917,Z 377.424,A -85,B 0,C 180,E1 22071.162,E2 22071.162} C_VEL
LIN {X 0,Y 487.488,Z 381.358,A -85,B 0,C 180,E1 22070.726,E2 22070.726} C_VEL
LIN {X 0,Y 489.193,Z 383.447,A -85,B 0,C 180,E1 22070.452,E2 22070.452} C_VEL
LIN {X 0,Y 500.642,Z 399.137,A -85,B 0,C 180,E1 22068.665,E2 22068.665} C_VEL
LIN {X 0,Y 510.582,Z 413.703,A -85,B 0,C 180,E1 22067.197,E2 22067.197} C_VEL
LIN {X 0,Y 505.831,Z 630.493,A -85,B 0,C 180,E1 22063.548,E2 22063.548} C_VEL
LIN {X 0,Y 504.038,Z 712.295,A -85,B 0,C 180,E1 22062.171,E2 22062.171} C_VEL
LIN {X 0,Y 502.902,Z 735.158,A -85,B 0,C 180,E1 22061.591,E2 22061.591} C_VEL
LIN {X 0,Y 501.436,Z 757.326,A -85,B 0,C 180,E1 22060.828,E2 22060.828} C_VEL
LIN {X 0,Y 499.623,Z 779.292,A -85,B 0,C 180,E1 22059.848,E2 22059.848} C_VEL
LIN {X 0,Y 497.527,Z 801.914,A -85,B 0,C 180,E1 22058.599,E2 22058.599} C_VEL
LIN {X 0,Y 495.198,Z 823.786,A -85,B 0,C 180,E1 22057.129,E2 22057.129} C_VEL
LIN {X 0,Y 492.957,Z 843.954,A -85,B 0,C 180,E1 22055.525,E2 22055.525} C_VEL
LIN {X 0,Y 490.721,Z 863.192,A -85,B 0,C 180,E1 22053.735,E2 22053.735} C_VEL
LIN {X 0,Y 488.558,Z 881.412,A -85,B 0,C 180,E1 22051.756,E2 22051.756} C_VEL
LIN {X 0,Y 486.587,Z 898.293,A -85,B 0,C 180,E1 22049.643,E2 22049.643} C_VEL
LIN {X 0,Y 484.789,Z 914.657,A -85,B 0,C 180,E1 22047.278,E2 22047.278} C_VEL
LIN {X 0,Y 483.342,Z 928.938,A -85,B 0,C 180,E1 22044.893,E2 22044.893} C_VEL
LIN {X 0,Y 482.102,Z 942.475,A -85,B 0,C 180,E1 22042.249,E2 22042.249} C_VEL
LIN {X 0,Y 481.242,Z 953.551,A -85,B 0,C 180,E1 22039.704,E2 22039.704} C_VEL
LIN {X 0,Y 480.644,Z 962.984,A -85,B 0,C 180,E1 22037.136,E2 22037.136} C_VEL
LIN {X 0,Y 480.26,Z 970.957,A -85,B 0,C 180,E1 22034.542,E2 22034.542} C_VEL
LIN {X 0,Y 480.05,Z 977.673,A -85,B 0,C 180,E1 22031.764,E2 22031.764} C_VEL
LIN {X 0,Y 479.94,Z 982.669,A -85,B 0,C 180,E1 22029,E2 22029} C_VEL
LIN {X 0,Y 479.893,Z 985.964,A -85,B 0,C 180,E1 22026.286,E2 22026.286} C_VEL
LIN {X 0,Y 479.889,Z 987.701,A -85,B 0,C 180,E1 22023.627,E2 22023.627} C_VEL
LIN {X 0,Y 479.915,Z 987.834,A -85,B 0,C 180,E1 22020.956,E2 22020.956} C_VEL
LIN {X 0,Y 479.91,Z 986.447,A -85,B 0,C 180,E1 22018.187,E2 22018.187} C_VEL
LIN {X 0,Y 479.925,Z 983.653,A -85,B 0,C 180,E1 22015.591,E2 22015.591} C_VEL
LIN {X 0,Y 480.003,Z 979.24,A -85,B 0,C 180,E1 22012.921,E2 22012.921} C_VEL
LIN {X 0,Y 480.209,Z 972.881,A -85,B 0,C 180,E1 22010.109,E2 22010.109} C_VEL
LIN {X 0,Y 480.567,Z 964.695,A -85,B 0,C 180,E1 22007.289,E2 22007.289} C_VEL
LIN {X 0,Y 481.147,Z 955.219,A -85,B 0,C 180,E1 22004.62,E2 22004.62} C_VEL
LIN {X 0,Y 482.019,Z 943.627,A -85,B 0,C 180,E1 22001.908,E2 22001.908} C_VEL
LIN {X 0,Y 483.201,Z 930.384,A -85,B 0,C 180,E1 21999.286,E2 21999.286} C_VEL
LIN {X 0,Y 484.658,Z 915.874,A -85,B 0,C 180,E1 21996.824,E2 21996.824} C_VEL
LIN {X 0,Y 486.453,Z 899.435,A -85,B 0,C 180,E1 21994.419,E2 21994.419} C_VEL
LIN {X 0,Y 488.444,Z 882.51,A -85,B 0,C 180,E1 21992.28,E2 21992.28} C_VEL
LIN {X 0,Y 490.669,Z 863.651,A -85,B 0,C 180,E1 21990.221,E2 21990.221} C_VEL
LIN {X 0,Y 492.942,Z 844.062,A -85,B 0,C 180,E1 21988.395,E2 21988.395} C_VEL
LIN {X 0,Y 495.159,Z 824.121,A -85,B 0,C 180,E1 21986.806,E2 21986.806} C_VEL
LIN {X 0,Y 497.47,Z 802.526,A -85,B 0,C 180,E1 21985.348,E2 21985.348} C_VEL
LIN {X 0,Y 499.537,Z 780.377,A -85,B 0,C 180,E1 21984.113,E2 21984.113} C_VEL
LIN {X 0,Y 501.404,Z 757.822,A -85,B 0,C 180,E1 21983.101,E2 21983.101} C_VEL
LIN {X 0,Y 502.871,Z 735.488,A -85,B 0,C 180,E1 21982.33,E2 21982.33} C_VEL
LIN {X 0,Y 503.996,Z 713.069,A -85,B 0,C 180,E1 21981.758,E2 21981.758} C_VEL
LIN {X 0,Y 505.453,Z 648.044,A -85,B 0,C 180,E1 21980.655,E2 21980.655} C_VEL
LIN {X 0,Y 509.948,Z 441.689,A -85,B 0,C 180,E1 21977.189,E2 21977.189} C_VEL
LIN {X 0,Y 510.494,Z 413.359,A -85,B 0,C 180,E1 21976.689,E2 21976.689} C_VEL
LIN {X 0,Y 498.857,Z 396.553,A -85,B 0,C 180,E1 21974.94,E2 21974.94} C_VEL
LIN {X 0,Y 491.509,Z 386.588,A -85,B 0,C 180,E1 21973.77,E2 21973.77} C_VEL
LIN {X 0,Y 488.098,Z 381.927,A -85,B 0,C 180,E1 21973.204,E2 21973.204} C_VEL
LIN {X 0,Y 485.329,Z 378.221,A -85,B 0,C 180,E1 21972.735,E2 21972.735} C_VEL
LIN {X 0,Y 484.451,Z 376.869,A -85,B 0,C 180,E1 21972.577,E2 21972.577} C_VEL
LIN {X 0,Y 481.911,Z 374.177,A -85,B 0,C 180,E1 21972.142,E2 21972.142} C_VEL
LIN {X 0,Y 480.994,Z 371.786,A -85,B 0,C 180,E1 21971.877,E2 21971.877} C_VEL
LIN {X 0,Y 480.89,Z 371.152,A -85,B 0,C 180,E1 21971.514,E2 21971.514} C_VEL
LIN {X 0,Y 480.885,Z 371.142,A -85,B 0,C 180,E1 21967.888,E2 21967.888} C_VEL
LIN {X 0,Y 480.885,Z 371.144,A -85,B 0,C 180,E1 21964.293,E2 21964.293} C_VEL
LIN {X 0,Y 480.884,Z 371.145,A -85,B 0,C 180,E1 21960.715,E2 21960.715} C_VEL
LIN {X 0,Y 480.879,Z 371.138,A -85,B 0,C 180,E1 21957.14,E2 21957.14} C_VEL
LIN {X 0,Y 480.868,Z 371.147,A -85,B 0,C 180,E1 21953.554,E2 21953.554} C_VEL
LIN {X 0,Y 480.886,Z 371.15,A -85,B 0,C 180,E1 21949.942,E2 21949.942} C_VEL
LIN {X 0,Y 480.894,Z 371.147,A -85,B 0,C 180,E1 21946.289,E2 21946.289} C_VEL
LIN {X 0,Y 480.868,Z 371.146,A -85,B 0,C 180,E1 21942.703,E2 21942.703} C_VEL
LIN {X 0,Y 480.846,Z 371.143,A -85,B 0,C 180,E1 21939.172,E2 21939.172} C_VEL
LIN {X 0,Y 480.873,Z 371.144,A -85,B 0,C 180,E1 21935.689,E2 21935.689} C_VEL
LIN {X 0,Y 480.889,Z 371.148,A -85,B 0,C 180,E1 21932.09,E2 21932.09} C_VEL
LIN {X 0,Y 480.829,Z 371.15,A -85,B 0,C 180,E1 21928.678,E2 21928.678} C_VEL
LIN {X 0,Y 480.824,Z 371.152,A -85,B 0,C 180,E1 21925.019,E2 21925.019} C_VEL
LIN {X 0,Y 480.908,Z 371.415,A -85,B 0,C 180,E1 21921.833,E2 21921.833} C_VEL
LIN {X 0,Y 482.195,Z 374.711,A -85,B 0,C 180,E1 21921.229,E2 21921.229} C_VEL
LIN {X 0,Y 483.596,Z 377.323,A -85,B 0,C 180,E1 21920.753,E2 21920.753} C_VEL
LIN {X 0,Y 486.057,Z 382.076,A -85,B 0,C 180,E1 21919.92,E2 21919.92} C_VEL
LIN {X 0,Y 489.116,Z 387.93,A -85,B 0,C 180,E1 21918.99,E2 21918.99} C_VEL
LIN {X 0,Y 499.282,Z 402.938,A -85,B 0,C 180,E1 21917.342,E2 21917.342} C_VEL
LIN {X 0,Y 510.805,Z 421.292,A -85,B 0,C 180,E1 21915.591,E2 21915.591} C_VEL
LIN {X 0,Y 506.249,Z 629.943,A -85,B 0,C 180,E1 21912.073,E2 21912.073} C_VEL
LIN {X 0,Y 503.945,Z 740.292,A -85,B 0,C 180,E1 21910.234,E2 21910.234} C_VEL
LIN {X 0,Y 502.83,Z 762.964,A -85,B 0,C 180,E1 21909.672,E2 21909.672} C_VEL
LIN {X 0,Y 501.535,Z 783.728,A -85,B 0,C 180,E1 21908.983,E2 21908.983} C_VEL
LIN {X 0,Y 499.801,Z 805.868,A -85,B 0,C 180,E1 21908.039,E2 21908.039} C_VEL
LIN {X 0,Y 497.916,Z 827.559,A -85,B 0,C 180,E1 21906.902,E2 21906.902} C_VEL
LIN {X 0,Y 495.917,Z 847.188,A -85,B 0,C 180,E1 21905.642,E2 21905.642} C_VEL
LIN {X 0,Y 493.809,Z 866.594,A -85,B 0,C 180,E1 21904.188,E2 21904.188} C_VEL
LIN {X 0,Y 491.541,Z 885.897,A -85,B 0,C 180,E1 21902.483,E2 21902.483} C_VEL
LIN {X 0,Y 489.378,Z 904.54,A -85,B 0,C 180,E1 21900.583,E2 21900.583} C_VEL
LIN {X 0,Y 487.385,Z 921.321,A -85,B 0,C 180,E1 21898.595,E2 21898.595} C_VEL
LIN {X 0,Y 485.468,Z 938.274,A -85,B 0,C 180,E1 21896.286,E2 21896.286} C_VEL
LIN {X 0,Y 483.959,Z 952.72,A -85,B 0,C 180,E1 21894.02,E2 21894.02} C_VEL
LIN {X 0,Y 482.633,Z 966.315,A -85,B 0,C 180,E1 21891.538,E2 21891.538} C_VEL
LIN {X 0,Y 481.637,Z 978.236,A -85,B 0,C 180,E1 21889.025,E2 21889.025} C_VEL
LIN {X 0,Y 480.932,Z 988.136,A -85,B 0,C 180,E1 21886.551,E2 21886.551} C_VEL
LIN {X 0,Y 480.425,Z 997.272,A -85,B 0,C 180,E1 21883.851,E2 21883.851} C_VEL
LIN {X 0,Y 480.142,Z 1003.948,A -85,B 0,C 180,E1 21881.413,E2 21881.413} C_VEL
LIN {X 0,Y 480,Z 1009.803,A -85,B 0,C 180,E1 21878.75,E2 21878.75} C_VEL
LIN {X 0,Y 479.928,Z 1013.955,A -85,B 0,C 180,E1 21876.103,E2 21876.103} C_VEL
LIN {X 0,Y 479.89,Z 1016.712,A -85,B 0,C 180,E1 21873.468,E2 21873.468} C_VEL
LIN {X 0,Y 479.891,Z 1017.826,A -85,B 0,C 180,E1 21870.959,E2 21870.959} C_VEL
LIN {X 0,Y 479.907,Z 1017.714,A -85,B 0,C 180,E1 21868.452,E2 21868.452} C_VEL
LIN {X 0,Y 479.911,Z 1015.959,A -85,B 0,C 180,E1 21865.702,E2 21865.702} C_VEL
LIN {X 0,Y 479.928,Z 1013.006,A -85,B 0,C 180,E1 21863.184,E2 21863.184} C_VEL
LIN {X 0,Y 480.02,Z 1008.345,A -85,B 0,C 180,E1 21860.533,E2 21860.533} C_VEL
LIN {X 0,Y 480.203,Z 1002.751,A -85,B 0,C 180,E1 21858.108,E2 21858.108} C_VEL
LIN {X 0,Y 480.575,Z 994.57,A -85,B 0,C 180,E1 21855.3,E2 21855.3} C_VEL
LIN {X 0,Y 481.099,Z 985.865,A -85,B 0,C 180,E1 21852.84,E2 21852.84} C_VEL
LIN {X 0,Y 481.91,Z 974.891,A -85,B 0,C 180,E1 21850.238,E2 21850.238} C_VEL
LIN {X 0,Y 483.014,Z 962.485,A -85,B 0,C 180,E1 21847.713,E2 21847.713} C_VEL
LIN {X 0,Y 484.401,Z 948.293,A -85,B 0,C 180,E1 21845.258,E2 21845.258} C_VEL
LIN {X 0,Y 486.159,Z 932.145,A -85,B 0,C 180,E1 21842.839,E2 21842.839} C_VEL
LIN {X 0,Y 487.975,Z 916.412,A -85,B 0,C 180,E1 21840.793,E2 21840.793} C_VEL
LIN {X 0,Y 490.044,Z 898.652,A -85,B 0,C 180,E1 21838.791,E2 21838.791} C_VEL
LIN {X 0,Y 492.24,Z 880.257,A -85,B 0,C 180,E1 21836.985,E2 21836.985} C_VEL
LIN {X 0,Y 494.406,Z 861.009,A -85,B 0,C 180,E1 21835.376,E2 21835.376} C_VEL
LIN {X 0,Y 496.59,Z 840.923,A -85,B 0,C 180,E1 21833.925,E2 21833.925} C_VEL
LIN {X 0,Y 498.517,Z 820.859,A -85,B 0,C 180,E1 21832.726,E2 21832.726} C_VEL
LIN {X 0,Y 500.452,Z 798.776,A -85,B 0,C 180,E1 21831.628,E2 21831.628} C_VEL
LIN {X 0,Y 501.967,Z 777.462,A -85,B 0,C 180,E1 21830.785,E2 21830.785} C_VEL
LIN {X 0,Y 503.357,Z 753.794,A -85,B 0,C 180,E1 21830.067,E2 21830.067} C_VEL
LIN {X 0,Y 504.261,Z 731.957,A -85,B 0,C 180,E1 21829.605,E2 21829.605} C_VEL
LIN {X 0,Y 508.648,Z 520.88,A -85,B 0,C 180,E1 21826.089,E2 21826.089} C_VEL
LIN {X 0,Y 510.748,Z 421.01,A -85,B 0,C 180,E1 21824.381,E2 21824.381} C_VEL
LIN {X 0,Y 497.111,Z 399.901,A -85,B 0,C 180,E1 21822.321,E2 21822.321} C_VEL
LIN {X 0,Y 489.154,Z 388.144,A -85,B 0,C 180,E1 21821.006,E2 21821.006} C_VEL
LIN {X 0,Y 484.822,Z 379.577,A -85,B 0,C 180,E1 21819.587,E2 21819.587} C_VEL
LIN {X 0,Y 482.329,Z 374.881,A -85,B 0,C 180,E1 21818.758,E2 21818.758} C_VEL
LIN {X 0,Y 480.894,Z 371.29,A -85,B 0,C 180,E1 21818.096,E2 21818.096} C_VEL
LIN {X 0,Y 480.832,Z 371.12,A -85,B 0,C 180,E1 21814.577,E2 21814.577} C_VEL
LIN {X 0,Y 480.808,Z 371.123,A -85,B 0,C 180,E1 21811.045,E2 21811.045} C_VEL
LIN {X 0,Y 480.848,Z 371.153,A -85,B 0,C 180,E1 21807.625,E2 21807.625} C_VEL
LIN {X 0,Y 480.845,Z 371.149,A -85,B 0,C 180,E1 21804.112,E2 21804.112} C_VEL
LIN {X 0,Y 480.81,Z 371.15,A -85,B 0,C 180,E1 21800.66,E2 21800.66} C_VEL
LIN {X 0,Y 480.838,Z 371.15,A -85,B 0,C 180,E1 21797.174,E2 21797.174} C_VEL
LIN {X 0,Y 480.849,Z 371.147,A -85,B 0,C 180,E1 21793.834,E2 21793.834} C_VEL
LIN {X 0,Y 480.817,Z 371.152,A -85,B 0,C 180,E1 21790.423,E2 21790.423} C_VEL
LIN {X 0,Y 480.85,Z 371.149,A -85,B 0,C 180,E1 21786.926,E2 21786.926} C_VEL
LIN {X 0,Y 480.865,Z 371.152,A -85,B 0,C 180,E1 21783.457,E2 21783.457} C_VEL
LIN {X 0,Y 480.825,Z 371.152,A -85,B 0,C 180,E1 21780,E2 21780} C_VEL
LIN {X 0,Y 480.84,Z 371.147,A -85,B 0,C 180,E1 21776.384,E2 21776.384} C_VEL
LIN {X 0,Y 480.893,Z 371.14,A -85,B 0,C 180,E1 21772.833,E2 21772.833} C_VEL
LIN {X 0,Y 480.85,Z 371.15,A -85,B 0,C 180,E1 21769.335,E2 21769.335} C_VEL
LIN {X 0,Y 480.836,Z 371.147,A -85,B 0,C 180,E1 21765.796,E2 21765.796} C_VEL
LIN {X 0,Y 480.878,Z 371.139,A -85,B 0,C 180,E1 21762.327,E2 21762.327} C_VEL
LIN {X 0,Y 480.875,Z 371.144,A -85,B 0,C 180,E1 21758.789,E2 21758.789} C_VEL
LIN {X 0,Y 480.842,Z 371.147,A -85,B 0,C 180,E1 21755.294,E2 21755.294} C_VEL
LIN {X 0,Y 480.857,Z 371.139,A -85,B 0,C 180,E1 21751.7,E2 21751.7} C_VEL
LIN {X 0,Y 480.895,Z 371.14,A -85,B 0,C 180,E1 21748.242,E2 21748.242} C_VEL
LIN {X 0,Y 480.86,Z 371.143,A -85,B 0,C 180,E1 21744.686,E2 21744.686} C_VEL
LIN {X 0,Y 480.854,Z 371.145,A -85,B 0,C 180,E1 21741.1,E2 21741.1} C_VEL
LIN {X 0,Y 480.884,Z 371.145,A -85,B 0,C 180,E1 21737.564,E2 21737.564} C_VEL
LIN {X 0,Y 480.891,Z 371.143,A -85,B 0,C 180,E1 21733.976,E2 21733.976} C_VEL
LIN {X 0,Y 480.863,Z 371.144,A -85,B 0,C 180,E1 21730.44,E2 21730.44} C_VEL
LIN {X 0,Y 480.865,Z 371.147,A -85,B 0,C 180,E1 21726.78,E2 21726.78} C_VEL
LIN {X 0,Y 480.889,Z 371.121,A -85,B 0,C 180,E1 21723.286,E2 21723.286} C_VEL
LIN {X 0,Y 480.892,Z 371.12,A -85,B 0,C 180,E1 21719.645,E2 21719.645} C_VEL
LIN {X 0,Y 480.872,Z 371.134,A -85,B 0,C 180,E1 21717.937,E2 21717.937} C_VEL
LIN {X 0,Y 479.906,Z 371.271,A -85,B 0,C 180,E1 21717.019,E2 21717.019} C_VEL
LIN {X 0,Y 473.362,Z 372.059,A -85,B 0,C 180,E1 21714.37,E2 21714.37} C_VEL
LIN {X 0,Y 472.94,Z 372.119,A -85,B 0,C 180,E1 21713.763,E2 21713.763} C_VEL
LIN {X 0,Y 472.988,Z 372.395,A -85,B 0,C 180,E1 21713.138,E2 21713.138} C_VEL
LIN {X 0,Y 473.379,Z 373.893,A -85,B 0,C 180,E1 21712.896,E2 21712.896} C_VEL
LIN {X 0,Y 475.261,Z 376.833,A -85,B 0,C 180,E1 21712.545,E2 21712.545} C_VEL
LIN {X 0,Y 477.067,Z 378.461,A -85,B 0,C 180,E1 21712.243,E2 21712.243} C_VEL
LIN {X 0,Y 479.614,Z 382.339,A -85,B 0,C 180,E1 21711.789,E2 21711.789} C_VEL
LIN {X 0,Y 481.403,Z 384.438,A -85,B 0,C 180,E1 21711.489,E2 21711.489} C_VEL
LIN {X 0,Y 493.397,Z 400.811,A -85,B 0,C 180,E1 21709.53,E2 21709.53} C_VEL
LIN {X 0,Y 504.886,Z 417.265,A -85,B 0,C 180,E1 21707.785,E2 21707.785} C_VEL
LIN {X 0,Y 499.791,Z 632.748,A -85,B 0,C 180,E1 21704.119,E2 21704.119} C_VEL
LIN {X 0,Y 497.896,Z 712.828,A -85,B 0,C 180,E1 21702.754,E2 21702.754} C_VEL
LIN {X 0,Y 496.684,Z 735.563,A -85,B 0,C 180,E1 21702.169,E2 21702.169} C_VEL
LIN {X 0,Y 495.161,Z 757.5,A -85,B 0,C 180,E1 21701.409,E2 21701.409} C_VEL
LIN {X 0,Y 493.28,Z 778.939,A -85,B 0,C 180,E1 21700.448,E2 21700.448} C_VEL
LIN {X 0,Y 491.128,Z 800.623,A -85,B 0,C 180,E1 21699.251,E2 21699.251} C_VEL
LIN {X 0,Y 488.844,Z 821.313,A -85,B 0,C 180,E1 21697.873,E2 21697.873} C_VEL
LIN {X 0,Y 486.356,Z 841.835,A -85,B 0,C 180,E1 21696.251,E2 21696.251} C_VEL
LIN {X 0,Y 483.922,Z 861.276,A -85,B 0,C 180,E1 21694.44,E2 21694.44} C_VEL
LIN {X 0,Y 481.538,Z 879.801,A -85,B 0,C 180,E1 21692.436,E2 21692.436} C_VEL
LIN {X 0,Y 479.352,Z 897.338,A -85,B 0,C 180,E1 21690.235,E2 21690.235} C_VEL
LIN {X 0,Y 477.457,Z 913.088,A -85,B 0,C 180,E1 21687.956,E2 21687.956} C_VEL
LIN {X 0,Y 475.833,Z 927.536,A -85,B 0,C 180,E1 21685.537,E2 21685.537} C_VEL
LIN {X 0,Y 474.504,Z 940.698,A -85,B 0,C 180,E1 21682.97,E2 21682.97} C_VEL
LIN {X 0,Y 473.518,Z 951.994,A -85,B 0,C 180,E1 21680.394,E2 21680.394} C_VEL
LIN {X 0,Y 472.789,Z 962.109,A -85,B 0,C 180,E1 21677.664,E2 21677.664} C_VEL
LIN {X 0,Y 472.344,Z 970.191,A -85,B 0,C 180,E1 21675.031,E2 21675.031} C_VEL
LIN {X 0,Y 472.083,Z 977.015,A -85,B 0,C 180,E1 21672.239,E2 21672.239} C_VEL
LIN {X 0,Y 471.966,Z 982.23,A -85,B 0,C 180,E1 21669.407,E2 21669.407} C_VEL
LIN {X 0,Y 471.894,Z 985.693,A -85,B 0,C 180,E1 21666.655,E2 21666.655} C_VEL
LIN {X 0,Y 471.89,Z 987.47,A -85,B 0,C 180,E1 21664.117,E2 21664.117} C_VEL
LIN {X 0,Y 471.908,Z 987.896,A -85,B 0,C 180,E1 21661.303,E2 21661.303} C_VEL
LIN {X 0,Y 471.907,Z 986.828,A -85,B 0,C 180,E1 21658.583,E2 21658.583} C_VEL
LIN {X 0,Y 471.912,Z 984.119,A -85,B 0,C 180,E1 21655.84,E2 21655.84} C_VEL
LIN {X 0,Y 471.985,Z 979.974,A -85,B 0,C 180,E1 21653.162,E2 21653.162} C_VEL
LIN {X 0,Y 472.188,Z 974.126,A -85,B 0,C 180,E1 21650.401,E2 21650.401} C_VEL
LIN {X 0,Y 472.532,Z 966.795,A -85,B 0,C 180,E1 21647.708,E2 21647.708} C_VEL
LIN {X 0,Y 473.071,Z 957.991,A -85,B 0,C 180,E1 21645.076,E2 21645.076} C_VEL
LIN {X 0,Y 473.906,Z 947.328,A -85,B 0,C 180,E1 21642.398,E2 21642.398} C_VEL
LIN {X 0,Y 475.093,Z 934.667,A -85,B 0,C 180,E1 21639.71,E2 21639.71} C_VEL
LIN {X 0,Y 476.621,Z 920.437,A -85,B 0,C 180,E1 21637.137,E2 21637.137} C_VEL
LIN {X 0,Y 478.436,Z 904.909,A -85,B 0,C 180,E1 21634.73,E2 21634.73} C_VEL
LIN {X 0,Y 480.505,Z 888.063,A -85,B 0,C 180,E1 21632.471,E2 21632.471} C_VEL
LIN {X 0,Y 482.885,Z 869.206,A -85,B 0,C 180,E1 21630.292,E2 21630.292} C_VEL
LIN {X 0,Y 485.335,Z 850.036,A -85,B 0,C 180,E1 21628.393,E2 21628.393} C_VEL
LIN {X 0,Y 487.84,Z 829.709,A -85,B 0,C 180,E1 21626.666,E2 21626.666} C_VEL
LIN {X 0,Y 490.351,Z 808.142,A -85,B 0,C 180,E1 21625.127,E2 21625.127} C_VEL
LIN {X 0,Y 492.523,Z 787.267,A -85,B 0,C 180,E1 21623.892,E2 21623.892} C_VEL
LIN {X 0,Y 494.514,Z 764.85,A -85,B 0,C 180,E1 21622.809,E2 21622.809} C_VEL
LIN {X 0,Y 496.239,Z 742.331,A -85,B 0,C 180,E1 21621.95,E2 21621.95} C_VEL
LIN {X 0,Y 497.501,Z 720.343,A -85,B 0,C 180,E1 21621.332,E2 21621.332} C_VEL
LIN {X 0,Y 498.43,Z 694.047,A -85,B 0,C 180,E1 21620.818,E2 21620.818} C_VEL
LIN {X 0,Y 503.195,Z 485.325,A -85,B 0,C 180,E1 21617.296,E2 21617.296} C_VEL
LIN {X 0,Y 504.784,Z 417.009,A -85,B 0,C 180,E1 21616.1,E2 21616.1} C_VEL
LIN {X 0,Y 491.914,Z 398.493,A -85,B 0,C 180,E1 21614.088,E2 21614.088} C_VEL
LIN {X 0,Y 484.139,Z 388.096,A -85,B 0,C 180,E1 21612.797,E2 21612.797} C_VEL
LIN {X 0,Y 480.606,Z 383.289,A -85,B 0,C 180,E1 21612.17,E2 21612.17} C_VEL
LIN {X 0,Y 477.737,Z 379.643,A -85,B 0,C 180,E1 21611.652,E2 21611.652} C_VEL
LIN {X 0,Y 476.736,Z 377.985,A -85,B 0,C 180,E1 21611.459,E2 21611.459} C_VEL
LIN {X 0,Y 474.1,Z 375.4,A -85,B 0,C 180,E1 21610.988,E2 21610.988} C_VEL
LIN {X 0,Y 473.03,Z 372.719,A -85,B 0,C 180,E1 21610.659,E2 21610.659} C_VEL
LIN {X 0,Y 472.948,Z 372.133,A -85,B 0,C 180,E1 21610.23,E2 21610.23} C_VEL
LIN {X 0,Y 472.94,Z 372.136,A -85,B 0,C 180,E1 21606.556,E2 21606.556} C_VEL
LIN {X 0,Y 472.946,Z 372.129,A -85,B 0,C 180,E1 21602.909,E2 21602.909} C_VEL
LIN {X 0,Y 472.939,Z 372.134,A -85,B 0,C 180,E1 21599.274,E2 21599.274} C_VEL
LIN {X 0,Y 472.934,Z 372.137,A -85,B 0,C 180,E1 21595.636,E2 21595.636} C_VEL
LIN {X 0,Y 472.95,Z 372.136,A -85,B 0,C 180,E1 21591.98,E2 21591.98} C_VEL
LIN {X 0,Y 472.954,Z 372.136,A -85,B 0,C 180,E1 21588.291,E2 21588.291} C_VEL
LIN {X 0,Y 472.94,Z 372.136,A -85,B 0,C 180,E1 21584.677,E2 21584.677} C_VEL
LIN {X 0,Y 472.912,Z 372.14,A -85,B 0,C 180,E1 21581.127,E2 21581.127} C_VEL
LIN {X 0,Y 472.92,Z 372.138,A -85,B 0,C 180,E1 21577.501,E2 21577.501} C_VEL
LIN {X 0,Y 472.95,Z 372.128,A -85,B 0,C 180,E1 21573.914,E2 21573.914} C_VEL
LIN {X 0,Y 472.903,Z 372.131,A -85,B 0,C 180,E1 21570.487,E2 21570.487} C_VEL
LIN {X 0,Y 472.887,Z 372.145,A -85,B 0,C 180,E1 21566.941,E2 21566.941} C_VEL
LIN {X 0,Y 472.91,Z 372.133,A -85,B 0,C 180,E1 21563.401,E2 21563.401} C_VEL
LIN {X 0,Y 472.966,Z 372.683,A -85,B 0,C 180,E1 21562.887,E2 21562.887} C_VEL
LIN {X 0,Y 474.271,Z 375.74,A -85,B 0,C 180,E1 21562.311,E2 21562.311} C_VEL
LIN {X 0,Y 475.413,Z 377.308,A -85,B 0,C 180,E1 21561.96,E2 21561.96} C_VEL
LIN {X 0,Y 480.382,Z 387.032,A -85,B 0,C 180,E1 21560.246,E2 21560.246} C_VEL
LIN {X 0,Y 490.422,Z 401.832,A -85,B 0,C 180,E1 21558.502,E2 21558.502} C_VEL
LIN {X 0,Y 502.14,Z 419.957,A -85,B 0,C 180,E1 21556.63,E2 21556.63} C_VEL
LIN {X 0,Y 505.082,Z 425.061,A -85,B 0,C 180,E1 21556.173,E2 21556.173} C_VEL
LIN {X 0,Y 500.173,Z 632.885,A -85,B 0,C 180,E1 21552.629,E2 21552.629} C_VEL
LIN {X 0,Y 497.756,Z 739.893,A -85,B 0,C 180,E1 21550.825,E2 21550.825} C_VEL
LIN {X 0,Y 496.554,Z 762.734,A -85,B 0,C 180,E1 21550.255,E2 21550.255} C_VEL
LIN {X 0,Y 495.13,Z 784.102,A -85,B 0,C 180,E1 21549.538,E2 21549.538} C_VEL
LIN {X 0,Y 493.233,Z 806.539,A -85,B 0,C 180,E1 21548.564,E2 21548.564} C_VEL
LIN {X 0,Y 491.216,Z 828.075,A -85,B 0,C 180,E1 21547.418,E2 21547.418} C_VEL
LIN {X 0,Y 489.016,Z 848.698,A -85,B 0,C 180,E1 21546.079,E2 21546.079} C_VEL
LIN {X 0,Y 486.77,Z 868.505,A -85,B 0,C 180,E1 21544.575,E2 21544.575} C_VEL
LIN {X 0,Y 484.403,Z 887.23,A -85,B 0,C 180,E1 21542.881,E2 21542.881} C_VEL
LIN {X 0,Y 481.898,Z 907.028,A -85,B 0,C 180,E1 21540.799,E2 21540.799} C_VEL
LIN {X 0,Y 479.817,Z 923.634,A -85,B 0,C 180,E1 21538.778,E2 21538.778} C_VEL
LIN {X 0,Y 477.904,Z 939.118,A -85,B 0,C 180,E1 21536.601,E2 21536.601} C_VEL
LIN {X 0,Y 476.282,Z 953.488,A -85,B 0,C 180,E1 21534.3,E2 21534.3} C_VEL
LIN {X 0,Y 474.85,Z 966.913,A -85,B 0,C 180,E1 21531.786,E2 21531.786} C_VEL
LIN {X 0,Y 473.727,Z 979.279,A -85,B 0,C 180,E1 21529.099,E2 21529.099} C_VEL
LIN {X 0,Y 472.983,Z 989.053,A -85,B 0,C 180,E1 21526.585,E2 21526.585} C_VEL
LIN {X 0,Y 472.429,Z 998.299,A -85,B 0,C 180,E1 21523.729,E2 21523.729} C_VEL
LIN {X 0,Y 472.139,Z 1004.857,A -85,B 0,C 180,E1 21521.238,E2 21521.238} C_VEL
LIN {X 0,Y 471.994,Z 1010.642,A -85,B 0,C 180,E1 21518.401,E2 21518.401} C_VEL
LIN {X 0,Y 471.918,Z 1014.433,A -85,B 0,C 180,E1 21515.84,E2 21515.84} C_VEL
LIN {X 0,Y 471.887,Z 1016.984,A -85,B 0,C 180,E1 21513.04,E2 21513.04} C_VEL
LIN {X 0,Y 471.884,Z 1017.871,A -85,B 0,C 180,E1 21510.732,E2 21510.732} C_VEL
LIN {X 0,Y 471.909,Z 1017.596,A -85,B 0,C 180,E1 21508.061,E2 21508.061} C_VEL
LIN {X 0,Y 471.906,Z 1015.732,A -85,B 0,C 180,E1 21505.386,E2 21505.386} C_VEL
LIN {X 0,Y 471.931,Z 1012.501,A -85,B 0,C 180,E1 21502.701,E2 21502.701} C_VEL
LIN {X 0,Y 472.034,Z 1007.836,A -85,B 0,C 180,E1 21500.125,E2 21500.125} C_VEL
LIN {X 0,Y 472.279,Z 1001.837,A -85,B 0,C 180,E1 21497.533,E2 21497.533} C_VEL
LIN {X 0,Y 472.702,Z 993.759,A -85,B 0,C 180,E1 21494.799,E2 21494.799} C_VEL
LIN {X 0,Y 473.341,Z 984.463,A -85,B 0,C 180,E1 21492.169,E2 21492.169} C_VEL
LIN {X 0,Y 474.267,Z 973.17,A -85,B 0,C 180,E1 21489.52,E2 21489.52} C_VEL
LIN {X 0,Y 475.581,Z 959.876,A -85,B 0,C 180,E1 21486.854,E2 21486.854} C_VEL
LIN {X 0,Y 477.053,Z 946.601,A -85,B 0,C 180,E1 21484.559,E2 21484.559} C_VEL
LIN {X 0,Y 478.905,Z 930.755,A -85,B 0,C 180,E1 21482.19,E2 21482.19} C_VEL
LIN {X 0,Y 480.974,Z 914.572,A -85,B 0,C 180,E1 21480.077,E2 21480.077} C_VEL
LIN {X 0,Y 483.19,Z 896.763,A -85,B 0,C 180,E1 21478.081,E2 21478.081} C_VEL
LIN {X 0,Y 485.619,Z 877.774,A -85,B 0,C 180,E1 21476.232,E2 21476.232} C_VEL
LIN {X 0,Y 487.724,Z 860.13,A -85,B 0,C 180,E1 21474.76,E2 21474.76} C_VEL
LIN {X 0,Y 490.04,Z 839.557,A -85,B 0,C 180,E1 21473.292,E2 21473.292} C_VEL
LIN {X 0,Y 491.999,Z 820.408,A -85,B 0,C 180,E1 21472.146,E2 21472.146} C_VEL
LIN {X 0,Y 494,Z 799.023,A -85,B 0,C 180,E1 21471.07,E2 21471.07} C_VEL
LIN {X 0,Y 495.656,Z 777.236,A -85,B 0,C 180,E1 21470.2,E2 21470.2} C_VEL
LIN {X 0,Y 497.163,Z 753.491,A -85,B 0,C 180,E1 21469.477,E2 21469.477} C_VEL
LIN {X 0,Y 498.113,Z 731.782,A -85,B 0,C 180,E1 21469.014,E2 21469.014} C_VEL
LIN {X 0,Y 502.846,Z 520.806,A -85,B 0,C 180,E1 21465.46,E2 21465.46} C_VEL
LIN {X 0,Y 505.077,Z 424.574,A -85,B 0,C 180,E1 21463.798,E2 21463.798} C_VEL
LIN {X 0,Y 491.676,Z 403.909,A -85,B 0,C 180,E1 21461.719,E2 21461.719} C_VEL
LIN {X 0,Y 484.078,Z 392.992,A -85,B 0,C 180,E1 21460.472,E2 21460.472} C_VEL
LIN {X 0,Y 480.649,Z 387.849,A -85,B 0,C 180,E1 21459.844,E2 21459.844} C_VEL
LIN {X 0,Y 476.743,Z 380.315,A -85,B 0,C 180,E1 21458.527,E2 21458.527} C_VEL
LIN {X 0,Y 474.713,Z 376.29,A -85,B 0,C 180,E1 21457.8,E2 21457.8} C_VEL
LIN {X 0,Y 473.021,Z 372.952,A -85,B 0,C 180,E1 21457.175,E2 21457.175} C_VEL
LIN {X 0,Y 472.892,Z 372.227,A -85,B 0,C 180,E1 21456.953,E2 21456.953} C_VEL
LIN {X 0,Y 472.879,Z 372.138,A -85,B 0,C 180,E1 21453.349,E2 21453.349} C_VEL
LIN {X 0,Y 472.934,Z 372.099,A -85,B 0,C 180,E1 21449.922,E2 21449.922} C_VEL
LIN {X 0,Y 472.879,Z 372.137,A -85,B 0,C 180,E1 21446.496,E2 21446.496} C_VEL
LIN {X 0,Y 472.871,Z 372.138,A -85,B 0,C 180,E1 21442.895,E2 21442.895} C_VEL
LIN {X 0,Y 472.92,Z 372.14,A -85,B 0,C 180,E1 21439.466,E2 21439.466} C_VEL
LIN {X 0,Y 472.913,Z 372.143,A -85,B 0,C 180,E1 21435.87,E2 21435.87} C_VEL
LIN {X 0,Y 472.88,Z 372.14,A -85,B 0,C 180,E1 21432.379,E2 21432.379} C_VEL
LIN {X 0,Y 472.891,Z 372.132,A -85,B 0,C 180,E1 21428.756,E2 21428.756} C_VEL
LIN {X 0,Y 472.938,Z 372.13,A -85,B 0,C 180,E1 21425.337,E2 21425.337} C_VEL
LIN {X 0,Y 472.894,Z 372.132,A -85,B 0,C 180,E1 21421.817,E2 21421.817} C_VEL
LIN {X 0,Y 472.889,Z 372.137,A -85,B 0,C 180,E1 21418.182,E2 21418.182} C_VEL
LIN {X 0,Y 472.928,Z 372.136,A -85,B 0,C 180,E1 21414.662,E2 21414.662} C_VEL
LIN {X 0,Y 472.932,Z 372.132,A -85,B 0,C 180,E1 21411.121,E2 21411.121} C_VEL
LIN {X 0,Y 472.897,Z 372.136,A -85,B 0,C 180,E1 21407.611,E2 21407.611} C_VEL
LIN {X 0,Y 472.912,Z 372.138,A -85,B 0,C 180,E1 21404.046,E2 21404.046} C_VEL
LIN {X 0,Y 472.952,Z 372.136,A -85,B 0,C 180,E1 21400.486,E2 21400.486} C_VEL
LIN {X 0,Y 472.92,Z 372.136,A -85,B 0,C 180,E1 21396.975,E2 21396.975} C_VEL
LIN {X 0,Y 472.907,Z 372.138,A -85,B 0,C 180,E1 21393.369,E2 21393.369} C_VEL
LIN {X 0,Y 472.934,Z 372.135,A -85,B 0,C 180,E1 21389.789,E2 21389.789} C_VEL
LIN {X 0,Y 472.956,Z 372.133,A -85,B 0,C 180,E1 21386.174,E2 21386.174} C_VEL
LIN {X 0,Y 472.923,Z 372.137,A -85,B 0,C 180,E1 21382.641,E2 21382.641} C_VEL
LIN {X 0,Y 472.916,Z 372.131,A -85,B 0,C 180,E1 21378.998,E2 21378.998} C_VEL
LIN {X 0,Y 472.942,Z 372.131,A -85,B 0,C 180,E1 21375.421,E2 21375.421} C_VEL
LIN {X 0,Y 472.955,Z 372.136,A -85,B 0,C 180,E1 21371.747,E2 21371.747} C_VEL
LIN {X 0,Y 472.937,Z 372.133,A -85,B 0,C 180,E1 21368.115,E2 21368.115} C_VEL
LIN {X 0,Y 472.922,Z 372.113,A -85,B 0,C 180,E1 21364.457,E2 21364.457} C_VEL
LIN {X 0,Y 472.938,Z 372.131,A -85,B 0,C 180,E1 21360.766,E2 21360.766} C_VEL
LIN {X 0,Y 472.954,Z 372.138,A -85,B 0,C 180,E1 21357.123,E2 21357.123} C_VEL
LIN {X 0,Y 472.94,Z 372.119,A -85,B 0,C 180,E1 21353.763,E2 21353.763} C_VEL
LIN {X 0,Y 473.335,Z 373.102,A -85,B 0,C 180,E1 21353.28,E2 21353.28} C_VEL
LIN {X 0,Y 474.501,Z 376.154,A -85,B 0,C 180,E1 21352.772,E2 21352.772} C_VEL
LIN {X 0,Y 476.584,Z 382.134,A -85,B 0,C 180,E1 21352.227,E2 21352.227} C_VEL
LIN {X 0,Y 480.288,Z 393.355,A -85,B 0,C 180,E1 21351.441,E2 21351.441} C_VEL
LIN {X 0,Y 482.632,Z 397.689,A -85,B 0,C 180,E1 21351.018,E2 21351.018} C_VEL
LIN {X 0,Y 492.737,Z 411.618,A -85,B 0,C 180,E1 21349.382,E2 21349.382} C_VEL
LIN {X 0,Y 499.219,Z 421.338,A -85,B 0,C 180,E1 21348.376,E2 21348.376} C_VEL
LIN {X 0,Y 493.773,Z 635.893,A -85,B 0,C 180,E1 21344.688,E2 21344.688} C_VEL
LIN {X 0,Y 491.811,Z 713.186,A -85,B 0,C 180,E1 21343.356,E2 21343.356} C_VEL
LIN {X 0,Y 490.539,Z 735.622,A -85,B 0,C 180,E1 21342.773,E2 21342.773} C_VEL
LIN {X 0,Y 488.937,Z 757.673,A -85,B 0,C 180,E1 21342.005,E2 21342.005} C_VEL
LIN {X 0,Y 486.882,Z 779.72,A -85,B 0,C 180,E1 21341.006,E2 21341.006} C_VEL
LIN {X 0,Y 484.495,Z 802.301,A -85,B 0,C 180,E1 21339.739,E2 21339.739} C_VEL
LIN {X 0,Y 481.969,Z 823.542,A -85,B 0,C 180,E1 21338.287,E2 21338.287} C_VEL
LIN {X 0,Y 479.329,Z 843.776,A -85,B 0,C 180,E1 21336.644,E2 21336.644} C_VEL
LIN {X 0,Y 476.66,Z 863.542,A -85,B 0,C 180,E1 21334.749,E2 21334.749} C_VEL
LIN {X 0,Y 474.128,Z 881.755,A -85,B 0,C 180,E1 21332.716,E2 21332.716} C_VEL
LIN {X 0,Y 471.919,Z 898.144,A -85,B 0,C 180,E1 21330.603,E2 21330.603} C_VEL
LIN {X 0,Y 469.879,Z 913.781,A -85,B 0,C 180,E1 21328.289,E2 21328.289} C_VEL
LIN {X 0,Y 468.147,Z 928.157,A -85,B 0,C 180,E1 21325.832,E2 21325.832} C_VEL
LIN {X 0,Y 466.658,Z 941.794,A -85,B 0,C 180,E1 21323.105,E2 21323.105} C_VEL
LIN {X 0,Y 465.603,Z 952.93,A -85,B 0,C 180,E1 21320.479,E2 21320.479} C_VEL
LIN {X 0,Y 464.829,Z 962.87,A -85,B 0,C 180,E1 21317.701,E2 21317.701} C_VEL
LIN {X 0,Y 464.36,Z 970.847,A -85,B 0,C 180,E1 21315.023,E2 21315.023} C_VEL
LIN {X 0,Y 464.086,Z 977.521,A -85,B 0,C 180,E1 21312.182,E2 21312.182} C_VEL
LIN {X 0,Y 463.96,Z 982.581,A -85,B 0,C 180,E1 21309.3,E2 21309.3} C_VEL
LIN {X 0,Y 463.891,Z 985.911,A -85,B 0,C 180,E1 21306.497,E2 21306.497} C_VEL
LIN {X 0,Y 463.885,Z 987.589,A -85,B 0,C 180,E1 21303.912,E2 21303.912} C_VEL
LIN {X 0,Y 463.91,Z 987.869,A -85,B 0,C 180,E1 21301.13,E2 21301.13} C_VEL
LIN {X 0,Y 463.909,Z 986.618,A -85,B 0,C 180,E1 21298.269,E2 21298.269} C_VEL
LIN {X 0,Y 463.925,Z 983.977,A -85,B 0,C 180,E1 21295.618,E2 21295.618} C_VEL
LIN {X 0,Y 464.016,Z 979.718,A -85,B 0,C 180,E1 21292.871,E2 21292.871} C_VEL
LIN {X 0,Y 464.24,Z 973.795,A -85,B 0,C 180,E1 21290.063,E2 21290.063} C_VEL
LIN {X 0,Y 464.64,Z 966.07,A -85,B 0,C 180,E1 21287.206,E2 21287.206} C_VEL
LIN {X 0,Y 465.281,Z 956.881,A -85,B 0,C 180,E1 21284.472,E2 21284.472} C_VEL
LIN {X 0,Y 466.269,Z 945.611,A -85,B 0,C 180,E1 21281.664,E2 21281.664} C_VEL
LIN {X 0,Y 467.647,Z 932.436,A -85,B 0,C 180,E1 21278.896,E2 21278.896} C_VEL
LIN {X 0,Y 469.347,Z 918.061,A -85,B 0,C 180,E1 21276.316,E2 21276.316} C_VEL
LIN {X 0,Y 471.338,Z 902.526,A -85,B 0,C 180,E1 21273.912,E2 21273.912} C_VEL
LIN {X 0,Y 473.649,Z 885.428,A -85,B 0,C 180,E1 21271.64,E2 21271.64} C_VEL
LIN {X 0,Y 476.087,Z 867.41,A -85,B 0,C 180,E1 21269.574,E2 21269.574} C_VEL
LIN {X 0,Y 478.809,Z 847.666,A -85,B 0,C 180,E1 21267.619,E2 21267.619} C_VEL
LIN {X 0,Y 481.441,Z 827.736,A -85,B 0,C 180,E1 21265.936,E2 21265.936} C_VEL
LIN {X 0,Y 483.984,Z 807.035,A -85,B 0,C 180,E1 21264.47,E2 21264.47} C_VEL
LIN {X 0,Y 486.243,Z 786.562,A -85,B 0,C 180,E1 21263.255,E2 21263.255} C_VEL
LIN {X 0,Y 488.279,Z 764.651,A -85,B 0,C 180,E1 21262.198,E2 21262.198} C_VEL
LIN {X 0,Y 490.116,Z 741.901,A -85,B 0,C 180,E1 21261.332,E2 21261.332} C_VEL
LIN {X 0,Y 491.369,Z 720.918,A -85,B 0,C 180,E1 21260.74,E2 21260.74} C_VEL
LIN {X 0,Y 492.339,Z 695.888,A -85,B 0,C 180,E1 21260.24,E2 21260.24} C_VEL
LIN {X 0,Y 497.475,Z 487.155,A -85,B 0,C 180,E1 21256.677,E2 21256.677} C_VEL
LIN {X 0,Y 499.164,Z 420.904,A -85,B 0,C 180,E1 21255.499,E2 21255.499} C_VEL
LIN {X 0,Y 487.671,Z 404.29,A -85,B 0,C 180,E1 21253.655,E2 21253.655} C_VEL
LIN {X 0,Y 479.984,Z 393.91,A -85,B 0,C 180,E1 21252.335,E2 21252.335} C_VEL
LIN {X 0,Y 476.556,Z 389.324,A -85,B 0,C 180,E1 21251.712,E2 21251.712} C_VEL
LIN {X 0,Y 472.917,Z 384.443,A -85,B 0,C 180,E1 21251.031,E2 21251.031} C_VEL
LIN {X 0,Y 470.034,Z 380.908,A -85,B 0,C 180,E1 21250.48,E2 21250.48} C_VEL
LIN {X 0,Y 468.965,Z 379.078,A -85,B 0,C 180,E1 21250.255,E2 21250.255} C_VEL
LIN {X 0,Y 466.212,Z 376.448,A -85,B 0,C 180,E1 21249.724,E2 21249.724} C_VEL
LIN {X 0,Y 465.135,Z 373.844,A -85,B 0,C 180,E1 21249.403,E2 21249.403} C_VEL
LIN {X 0,Y 465.006,Z 373.145,A -85,B 0,C 180,E1 21249.031,E2 21249.031} C_VEL
LIN {X 0,Y 465.007,Z 373.117,A -85,B 0,C 180,E1 21245.397,E2 21245.397} C_VEL
LIN {X 0,Y 465.001,Z 373.124,A -85,B 0,C 180,E1 21241.726,E2 21241.726} C_VEL
LIN {X 0,Y 465.01,Z 373.121,A -85,B 0,C 180,E1 21238.152,E2 21238.152} C_VEL
LIN {X 0,Y 465.01,Z 373.115,A -85,B 0,C 180,E1 21234.448,E2 21234.448} C_VEL
LIN {X 0,Y 465.003,Z 373.125,A -85,B 0,C 180,E1 21230.845,E2 21230.845} C_VEL
LIN {X 0,Y 464.982,Z 373.128,A -85,B 0,C 180,E1 21227.204,E2 21227.204} C_VEL
LIN {X 0,Y 464.986,Z 373.127,A -85,B 0,C 180,E1 21223.549,E2 21223.549} C_VEL
LIN {X 0,Y 465.015,Z 373.119,A -85,B 0,C 180,E1 21219.993,E2 21219.993} C_VEL
LIN {X 0,Y 464.99,Z 373.118,A -85,B 0,C 180,E1 21216.425,E2 21216.425} C_VEL
LIN {X 0,Y 464.959,Z 373.124,A -85,B 0,C 180,E1 21212.878,E2 21212.878} C_VEL
LIN {X 0,Y 464.96,Z 373.131,A -85,B 0,C 180,E1 21209.217,E2 21209.217} C_VEL
LIN {X 0,Y 464.996,Z 373.118,A -85,B 0,C 180,E1 21205.663,E2 21205.663} C_VEL
LIN {X 0,Y 465.008,Z 373.422,A -85,B 0,C 180,E1 21204.16,E2 21204.16} C_VEL
LIN {X 0,Y 466.516,Z 376.938,A -85,B 0,C 180,E1 21203.429,E2 21203.429} C_VEL
LIN {X 0,Y 467.569,Z 378.563,A -85,B 0,C 180,E1 21203.067,E2 21203.067} C_VEL
LIN {X 0,Y 469.525,Z 382.279,A -85,B 0,C 180,E1 21202.326,E2 21202.326} C_VEL
LIN {X 0,Y 472,Z 386.802,A -85,B 0,C 180,E1 21201.519,E2 21201.519} C_VEL
LIN {X 0,Y 480.245,Z 398.613,A -85,B 0,C 180,E1 21199.98,E2 21199.98} C_VEL
LIN {X 0,Y 490.805,Z 414.469,A -85,B 0,C 180,E1 21198.171,E2 21198.171} C_VEL
LIN {X 0,Y 499.439,Z 428.675,A -85,B 0,C 180,E1 21196.774,E2 21196.774} C_VEL
LIN {X 0,Y 494.166,Z 635.05,A -85,B 0,C 180,E1 21193.213,E2 21193.213} C_VEL
LIN {X 0,Y 491.617,Z 739.711,A -85,B 0,C 180,E1 21191.427,E2 21191.427} C_VEL
LIN {X 0,Y 490.323,Z 762.611,A -85,B 0,C 180,E1 21190.85,E2 21190.85} C_VEL
LIN {X 0,Y 488.748,Z 784.848,A -85,B 0,C 180,E1 21190.095,E2 21190.095} C_VEL
LIN {X 0,Y 486.774,Z 806.559,A -85,B 0,C 180,E1 21189.135,E2 21189.135} C_VEL
LIN {X 0,Y 484.63,Z 827.855,A -85,B 0,C 180,E1 21187.991,E2 21187.991} C_VEL
LIN {X 0,Y 482.295,Z 848.294,A -85,B 0,C 180,E1 21186.65,E2 21186.65} C_VEL
LIN {X 0,Y 479.883,Z 868.447,A -85,B 0,C 180,E1 21185.107,E2 21185.107} C_VEL
LIN {X 0,Y 477.449,Z 887.165,A -85,B 0,C 180,E1 21183.422,E2 21183.422} C_VEL
LIN {X 0,Y 475.039,Z 905.221,A -85,B 0,C 180,E1 21181.523,E2 21181.523} C_VEL
LIN {X 0,Y 472.777,Z 921.607,A -85,B 0,C 180,E1 21179.525,E2 21179.525} C_VEL
LIN {X 0,Y 470.58,Z 938.271,A -85,B 0,C 180,E1 21177.185,E2 21177.185} C_VEL
LIN {X 0,Y 468.781,Z 952.716,A -85,B 0,C 180,E1 21174.849,E2 21174.849} C_VEL
LIN {X 0,Y 467.266,Z 965.794,A -85,B 0,C 180,E1 21172.392,E2 21172.392} C_VEL
LIN {X 0,Y 466.081,Z 977.711,A -85,B 0,C 180,E1 21169.816,E2 21169.816} C_VEL
LIN {X 0,Y 465.172,Z 988.134,A -85,B 0,C 180,E1 21167.129,E2 21167.129} C_VEL
LIN {X 0,Y 464.551,Z 997.273,A -85,B 0,C 180,E1 21164.334,E2 21164.334} C_VEL
LIN {X 0,Y 464.214,Z 1003.947,A -85,B 0,C 180,E1 21161.811,E2 21161.811} C_VEL
LIN {X 0,Y 464.025,Z 1009.803,A -85,B 0,C 180,E1 21159.053,E2 21159.053} C_VEL
LIN {X 0,Y 463.941,Z 1013.955,A -85,B 0,C 180,E1 21156.314,E2 21156.314} C_VEL
LIN {X 0,Y 463.895,Z 1016.711,A -85,B 0,C 180,E1 21153.587,E2 21153.587} C_VEL
LIN {X 0,Y 463.892,Z 1017.826,A -85,B 0,C 180,E1 21150.992,E2 21150.992} C_VEL
LIN {X 0,Y 463.907,Z 1017.714,A -85,B 0,C 180,E1 21148.398,E2 21148.398} C_VEL
LIN {X 0,Y 463.908,Z 1015.959,A -85,B 0,C 180,E1 21145.554,E2 21145.554} C_VEL
LIN {X 0,Y 463.927,Z 1013.165,A -85,B 0,C 180,E1 21143.072,E2 21143.072} C_VEL
LIN {X 0,Y 464.039,Z 1008.345,A -85,B 0,C 180,E1 21140.204,E2 21140.204} C_VEL
LIN {X 0,Y 464.273,Z 1002.753,A -85,B 0,C 180,E1 21137.694,E2 21137.694} C_VEL
LIN {X 0,Y 464.734,Z 994.568,A -85,B 0,C 180,E1 21134.787,E2 21134.787} C_VEL
LIN {X 0,Y 465.406,Z 985.404,A -85,B 0,C 180,E1 21132.113,E2 21132.113} C_VEL
LIN {X 0,Y 466.389,Z 974.315,A -85,B 0,C 180,E1 21129.42,E2 21129.42} C_VEL
LIN {X 0,Y 467.741,Z 961.776,A -85,B 0,C 180,E1 21126.806,E2 21126.806} C_VEL
LIN {X 0,Y 469.336,Z 948.14,A -85,B 0,C 180,E1 21124.381,E2 21124.381} C_VEL
LIN {X 0,Y 471.427,Z 931.679,A -85,B 0,C 180,E1 21121.847,E2 21121.847} C_VEL
LIN {X 0,Y 473.624,Z 915.579,A -85,B 0,C 180,E1 21119.703,E2 21119.703} C_VEL
LIN {X 0,Y 475.99,Z 898.039,A -85,B 0,C 180,E1 21117.689,E2 21117.689} C_VEL
LIN {X 0,Y 478.181,Z 881.826,A -85,B 0,C 180,E1 21116.069,E2 21116.069} C_VEL
LIN {X 0,Y 480.654,Z 862.189,A -85,B 0,C 180,E1 21114.383,E2 21114.383} C_VEL
LIN {X 0,Y 483.102,Z 842.07,A -85,B 0,C 180,E1 21112.899,E2 21112.899} C_VEL
LIN {X 0,Y 485.41,Z 821.1,A -85,B 0,C 180,E1 21111.615,E2 21111.615} C_VEL
LIN {X 0,Y 487.539,Z 799.994,A -85,B 0,C 180,E1 21110.53,E2 21110.53} C_VEL
LIN {X 0,Y 489.377,Z 777.317,A -85,B 0,C 180,E1 21109.612,E2 21109.612} C_VEL
LIN {X 0,Y 490.987,Z 753.809,A -85,B 0,C 180,E1 21108.886,E2 21108.886} C_VEL
LIN {X 0,Y 492.003,Z 732.067,A -85,B 0,C 180,E1 21108.416,E2 21108.416} C_VEL
LIN {X 0,Y 497.093,Z 521.236,A -85,B 0,C 180,E1 21104.824,E2 21104.824} C_VEL
LIN {X 0,Y 499.393,Z 428.2,A -85,B 0,C 180,E1 21103.194,E2 21103.194} C_VEL
LIN {X 0,Y 487.091,Z 409.175,A -85,B 0,C 180,E1 21101.237,E2 21101.237} C_VEL
LIN {X 0,Y 476.686,Z 394.013,A -85,B 0,C 180,E1 21099.46,E2 21099.46} C_VEL
LIN {X 0,Y 472.251,Z 387.624,A -85,B 0,C 180,E1 21098.633,E2 21098.633} C_VEL
LIN {X 0,Y 469.06,Z 381.705,A -85,B 0,C 180,E1 21097.546,E2 21097.546} C_VEL
LIN {X 0,Y 466.73,Z 377.245,A -85,B 0,C 180,E1 21096.704,E2 21096.704} C_VEL
LIN {X 0,Y 465.036,Z 373.46,A -85,B 0,C 180,E1 21095.973,E2 21095.973} C_VEL
LIN {X 0,Y 464.956,Z 373.094,A -85,B 0,C 180,E1 21094.561,E2 21094.561} C_VEL
LIN {X 0,Y 464.932,Z 373.096,A -85,B 0,C 180,E1 21091.073,E2 21091.073} C_VEL
LIN {X 0,Y 464.961,Z 373.131,A -85,B 0,C 180,E1 21087.538,E2 21087.538} C_VEL
LIN {X 0,Y 464.982,Z 373.122,A -85,B 0,C 180,E1 21083.966,E2 21083.966} C_VEL
LIN {X 0,Y 464.936,Z 373.126,A -85,B 0,C 180,E1 21080.52,E2 21080.52} C_VEL
LIN {X 0,Y 464.943,Z 373.131,A -85,B 0,C 180,E1 21076.876,E2 21076.876} C_VEL
LIN {X 0,Y 465,Z 373.127,A -85,B 0,C 180,E1 21073.428,E2 21073.428} C_VEL
LIN {X 0,Y 464.97,Z 373.131,A -85,B 0,C 180,E1 21069.78,E2 21069.78} C_VEL
LIN {X 0,Y 464.944,Z 373.128,A -85,B 0,C 180,E1 21066.296,E2 21066.296} C_VEL
LIN {X 0,Y 464.967,Z 373.12,A -85,B 0,C 180,E1 21062.711,E2 21062.711} C_VEL
LIN {X 0,Y 465.01,Z 373.118,A -85,B 0,C 180,E1 21059.137,E2 21059.137} C_VEL
LIN {X 0,Y 464.963,Z 373.123,A -85,B 0,C 180,E1 21055.56,E2 21055.56} C_VEL
LIN {X 0,Y 464.954,Z 373.119,A -85,B 0,C 180,E1 21051.964,E2 21051.964} C_VEL
LIN {X 0,Y 464.991,Z 373.119,A -85,B 0,C 180,E1 21048.464,E2 21048.464} C_VEL
LIN {X 0,Y 465.006,Z 373.118,A -85,B 0,C 180,E1 21044.871,E2 21044.871} C_VEL
LIN {X 0,Y 464.966,Z 373.119,A -85,B 0,C 180,E1 21041.312,E2 21041.312} C_VEL
LIN {X 0,Y 464.966,Z 373.123,A -85,B 0,C 180,E1 21037.603,E2 21037.603} C_VEL
LIN {X 0,Y 465.007,Z 373.122,A -85,B 0,C 180,E1 21034.119,E2 21034.119} C_VEL
LIN {X 0,Y 465.007,Z 373.121,A -85,B 0,C 180,E1 21030.501,E2 21030.501} C_VEL
LIN {X 0,Y 464.975,Z 373.127,A -85,B 0,C 180,E1 21026.894,E2 21026.894} C_VEL
LIN {X 0,Y 464.979,Z 373.126,A -85,B 0,C 180,E1 21023.288,E2 21023.288} C_VEL
LIN {X 0,Y 465.015,Z 373.118,A -85,B 0,C 180,E1 21019.669,E2 21019.669} C_VEL
LIN {X 0,Y 465.011,Z 373.117,A -85,B 0,C 180,E1 21016.011,E2 21016.011} C_VEL
LIN {X 0,Y 464.984,Z 373.119,A -85,B 0,C 180,E1 21012.462,E2 21012.462} C_VEL
LIN {X 0,Y 464.983,Z 373.127,A -85,B 0,C 180,E1 21008.73,E2 21008.73} C_VEL
LIN {X 0,Y 465.008,Z 373.11,A -85,B 0,C 180,E1 21005.181,E2 21005.181} C_VEL
LIN {X 0,Y 465.014,Z 373.126,A -85,B 0,C 180,E1 21001.494,E2 21001.494} C_VEL
LIN {X 0,Y 465.002,Z 373.11,A -85,B 0,C 180,E1 20997.808,E2 20997.808} C_VEL
LIN {X 0,Y 465.011,Z 373.256,A -85,B 0,C 180,E1 20994.378,E2 20994.378} C_VEL
LIN {X 0,Y 465.337,Z 374.644,A -85,B 0,C 180,E1 20994.101,E2 20994.101} C_VEL
LIN {X 0,Y 467.255,Z 377.747,A -85,B 0,C 180,E1 20993.717,E2 20993.717} C_VEL
LIN {X 0,Y 469.208,Z 379.504,A -85,B 0,C 180,E1 20993.377,E2 20993.377} C_VEL
LIN {X 0,Y 471.826,Z 383.474,A -85,B 0,C 180,E1 20992.891,E2 20992.891} C_VEL
LIN {X 0,Y 473.672,Z 385.553,A -85,B 0,C 180,E1 20992.571,E2 20992.571} C_VEL
LIN {X 0,Y 477.093,Z 389.919,A -85,B 0,C 180,E1 20991.972,E2 20991.972} C_VEL
LIN {X 0,Y 482.632,Z 397.689,A -85,B 0,C 180,E1 20991.018,E2 20991.018} C_VEL
LIN {X 0,Y 484.465,Z 401.663,A -85,B 0,C 180,E1 20990.68,E2 20990.68} C_VEL
LIN {X 0,Y 487.346,Z 414.649,A -85,B 0,C 180,E1 20990.009,E2 20990.009} C_VEL
LIN {X 0,Y 488.967,Z 418.075,A -85,B 0,C 180,E1 20989.724,E2 20989.724} C_VEL
LIN {X 0,Y 493.61,Z 425.113,A -85,B 0,C 180,E1 20988.985,E2 20988.985} C_VEL
LIN {X 0,Y 487.82,Z 638.544,A -85,B 0,C 180,E1 20985.28,E2 20985.28} C_VEL
LIN {X 0,Y 485.785,Z 713.313,A -85,B 0,C 180,E1 20983.976,E2 20983.976} C_VEL
LIN {X 0,Y 484.457,Z 735.565,A -85,B 0,C 180,E1 20983.395,E2 20983.395} C_VEL
LIN {X 0,Y 482.829,Z 757.1,A -85,B 0,C 180,E1 20982.646,E2 20982.646} C_VEL
LIN {X 0,Y 480.78,Z 778.18,A -85,B 0,C 180,E1 20981.695,E2 20981.695} C_VEL
LIN {X 0,Y 478.455,Z 799.323,A -85,B 0,C 180,E1 20980.532,E2 20980.532} C_VEL
LIN {X 0,Y 475.811,Z 820.488,A -85,B 0,C 180,E1 20979.109,E2 20979.109} C_VEL
LIN {X 0,Y 473.016,Z 841.046,A -85,B 0,C 180,E1 20977.465,E2 20977.465} C_VEL
LIN {X 0,Y 470.154,Z 860.624,A -85,B 0,C 180,E1 20975.61,E2 20975.61} C_VEL
LIN {X 0,Y 467.4,Z 879.146,A -85,B 0,C 180,E1 20973.553,E2 20973.553} C_VEL
LIN {X 0,Y 464.873,Z 896.323,A -85,B 0,C 180,E1 20971.352,E2 20971.352} C_VEL
LIN {X 0,Y 462.644,Z 912.214,A -85,B 0,C 180,E1 20969.006,E2 20969.006} C_VEL
LIN {X 0,Y 460.644,Z 927.426,A -85,B 0,C 180,E1 20966.387,E2 20966.387} C_VEL
LIN {X 0,Y 459.067,Z 940.546,A -85,B 0,C 180,E1 20963.744,E2 20963.744} C_VEL
LIN {X 0,Y 457.833,Z 952.372,A -85,B 0,C 180,E1 20960.95,E2 20960.95} C_VEL
LIN {X 0,Y 456.935,Z 962.815,A -85,B 0,C 180,E1 20957.999,E2 20957.999} C_VEL
LIN {X 0,Y 456.422,Z 970.792,A -85,B 0,C 180,E1 20955.276,E2 20955.276} C_VEL
LIN {X 0,Y 456.11,Z 977.469,A -85,B 0,C 180,E1 20952.388,E2 20952.388} C_VEL
LIN {X 0,Y 455.971,Z 982.554,A -85,B 0,C 180,E1 20949.445,E2 20949.445} C_VEL
LIN {X 0,Y 455.893,Z 985.884,A -85,B 0,C 180,E1 20946.608,E2 20946.608} C_VEL
LIN {X 0,Y 455.886,Z 987.572,A -85,B 0,C 180,E1 20943.979,E2 20943.979} C_VEL
LIN {X 0,Y 455.909,Z 987.874,A -85,B 0,C 180,E1 20941.149,E2 20941.149} C_VEL
LIN {X 0,Y 455.909,Z 986.706,A -85,B 0,C 180,E1 20938.314,E2 20938.314} C_VEL
LIN {X 0,Y 455.931,Z 984.018,A -85,B 0,C 180,E1 20935.539,E2 20935.539} C_VEL
LIN {X 0,Y 456.032,Z 979.767,A -85,B 0,C 180,E1 20932.74,E2 20932.74} C_VEL
LIN {X 0,Y 456.266,Z 973.88,A -85,B 0,C 180,E1 20929.886,E2 20929.886} C_VEL
LIN {X 0,Y 456.686,Z 966.461,A -85,B 0,C 180,E1 20927.083,E2 20927.083} C_VEL
LIN {X 0,Y 457.355,Z 957.591,A -85,B 0,C 180,E1 20924.364,E2 20924.364} C_VEL
LIN {X 0,Y 458.397,Z 946.6,A -85,B 0,C 180,E1 20921.536,E2 20921.536} C_VEL
LIN {X 0,Y 459.779,Z 934.384,A -85,B 0,C 180,E1 20918.871,E2 20918.871} C_VEL
LIN {X 0,Y 461.601,Z 919.975,A -85,B 0,C 180,E1 20916.188,E2 20916.188} C_VEL
LIN {X 0,Y 463.755,Z 904.141,A -85,B 0,C 180,E1 20913.669,E2 20913.669} C_VEL
LIN {X 0,Y 466.236,Z 887.112,A -85,B 0,C 180,E1 20911.336,E2 20911.336} C_VEL
LIN {X 0,Y 468.967,Z 868.702,A -85,B 0,C 180,E1 20909.155,E2 20909.155} C_VEL
LIN {X 0,Y 471.872,Z 849.126,A -85,B 0,C 180,E1 20907.17,E2 20907.17} C_VEL
LIN {X 0,Y 474.532,Z 830.128,A -85,B 0,C 180,E1 20905.531,E2 20905.531} C_VEL
LIN {X 0,Y 477.346,Z 808.716,A -85,B 0,C 180,E1 20903.977,E2 20903.977} C_VEL
LIN {X 0,Y 479.584,Z 789.657,A -85,B 0,C 180,E1 20902.817,E2 20902.817} C_VEL
LIN {X 0,Y 481.897,Z 766.776,A -85,B 0,C 180,E1 20901.674,E2 20901.674} C_VEL
LIN {X 0,Y 483.81,Z 744.659,A -85,B 0,C 180,E1 20900.802,E2 20900.802} C_VEL
LIN {X 0,Y 485.233,Z 722.611,A -85,B 0,C 180,E1 20900.16,E2 20900.16} C_VEL
LIN {X 0,Y 486.26,Z 699.226,A -85,B 0,C 180,E1 20899.672,E2 20899.672} C_VEL
LIN {X 0,Y 491.767,Z 491.093,A -85,B 0,C 180,E1 20896.079,E2 20896.079} C_VEL
LIN {X 0,Y 493.656,Z 424.708,A -85,B 0,C 180,E1 20894.89,E2 20894.89} C_VEL
LIN {X 0,Y 480.734,Z 406.162,A -85,B 0,C 180,E1 20892.737,E2 20892.737} C_VEL
LIN {X 0,Y 472.746,Z 395.486,A -85,B 0,C 180,E1 20891.282,E2 20891.282} C_VEL
LIN {X 0,Y 469.148,Z 390.735,A -85,B 0,C 180,E1 20890.593,E2 20890.593} C_VEL
LIN {X 0,Y 466.015,Z 386.374,A -85,B 0,C 180,E1 20889.958,E2 20889.958} C_VEL
LIN {X 0,Y 462.519,Z 382.437,A -85,B 0,C 180,E1 20889.253,E2 20889.253} C_VEL
LIN {X 0,Y 461.303,Z 380.23,A -85,B 0,C 180,E1 20888.979,E2 20888.979} C_VEL
LIN {X 0,Y 458.498,Z 377.778,A -85,B 0,C 180,E1 20888.402,E2 20888.402} C_VEL
LIN {X 0,Y 457.247,Z 375.047,A -85,B 0,C 180,E1 20888.045,E2 20888.045} C_VEL
LIN {X 0,Y 457.073,Z 374.146,A -85,B 0,C 180,E1 20887.669,E2 20887.669} C_VEL
LIN {X 0,Y 457.068,Z 374.117,A -85,B 0,C 180,E1 20883.889,E2 20883.889} C_VEL
LIN {X 0,Y 457.081,Z 374.103,A -85,B 0,C 180,E1 20880.126,E2 20880.126} C_VEL
LIN {X 0,Y 457.071,Z 374.108,A -85,B 0,C 180,E1 20876.363,E2 20876.363} C_VEL
LIN {X 0,Y 457.079,Z 374.114,A -85,B 0,C 180,E1 20872.585,E2 20872.585} C_VEL
LIN {X 0,Y 457.056,Z 374.113,A -85,B 0,C 180,E1 20868.901,E2 20868.901} C_VEL
LIN {X 0,Y 457.04,Z 374.117,A -85,B 0,C 180,E1 20865.236,E2 20865.236} C_VEL
LIN {X 0,Y 457.053,Z 374.115,A -85,B 0,C 180,E1 20861.639,E2 20861.639} C_VEL
LIN {X 0,Y 457.085,Z 374.111,A -85,B 0,C 180,E1 20858.035,E2 20858.035} C_VEL
LIN {X 0,Y 457.051,Z 374.112,A -85,B 0,C 180,E1 20854.333,E2 20854.333} C_VEL
LIN {X 0,Y 457.015,Z 374.109,A -85,B 0,C 180,E1 20850.799,E2 20850.799} C_VEL
LIN {X 0,Y 457.016,Z 374.119,A -85,B 0,C 180,E1 20847.142,E2 20847.142} C_VEL
LIN {X 0,Y 457.08,Z 374.412,A -85,B 0,C 180,E1 20845.463,E2 20845.463} C_VEL
LIN {X 0,Y 458.52,Z 377.903,A -85,B 0,C 180,E1 20844.7,E2 20844.7} C_VEL
LIN {X 0,Y 459.885,Z 380.008,A -85,B 0,C 180,E1 20844.193,E2 20844.193} C_VEL
LIN {X 0,Y 462.578,Z 385.145,A -85,B 0,C 180,E1 20843.144,E2 20843.144} C_VEL
LIN {X 0,Y 469.834,Z 395.336,A -85,B 0,C 180,E1 20841.64,E2 20841.64} C_VEL
LIN {X 0,Y 476.794,Z 405.284,A -85,B 0,C 180,E1 20840.326,E2 20840.326} C_VEL
LIN {X 0,Y 487.106,Z 421.077,A -85,B 0,C 180,E1 20838.51,E2 20838.51} C_VEL
LIN {X 0,Y 493.859,Z 432.249,A -85,B 0,C 180,E1 20837.389,E2 20837.389} C_VEL
LIN {X 0,Y 488.268,Z 635.21,A -85,B 0,C 180,E1 20833.845,E2 20833.845} C_VEL
LIN {X 0,Y 485.541,Z 739.421,A -85,B 0,C 180,E1 20832.045,E2 20832.045} C_VEL
LIN {X 0,Y 484.149,Z 762.449,A -85,B 0,C 180,E1 20831.462,E2 20831.462} C_VEL
LIN {X 0,Y 482.504,Z 784.326,A -85,B 0,C 180,E1 20830.713,E2 20830.713} C_VEL
LIN {X 0,Y 480.434,Z 805.929,A -85,B 0,C 180,E1 20829.753,E2 20829.753} C_VEL
LIN {X 0,Y 478.189,Z 826.903,A -85,B 0,C 180,E1 20828.622,E2 20828.622} C_VEL
LIN {X 0,Y 475.662,Z 847.593,A -85,B 0,C 180,E1 20827.259,E2 20827.259} C_VEL
LIN {X 0,Y 473.079,Z 867.935,A -85,B 0,C 180,E1 20825.688,E2 20825.688} C_VEL
LIN {X 0,Y 470.48,Z 886.669,A -85,B 0,C 180,E1 20823.984,E2 20823.984} C_VEL
LIN {X 0,Y 467.807,Z 905.983,A -85,B 0,C 180,E1 20821.95,E2 20821.95} C_VEL
LIN {X 0,Y 465.85,Z 919.579,A -85,B 0,C 180,E1 20820.293,E2 20820.293} C_VEL
LIN {X 0,Y 463.545,Z 935.732,A -85,B 0,C 180,E1 20818.052,E2 20818.052} C_VEL
LIN {X 0,Y 461.526,Z 950.403,A -85,B 0,C 180,E1 20815.679,E2 20815.679} C_VEL
LIN {X 0,Y 459.761,Z 964.522,A -85,B 0,C 180,E1 20813.048,E2 20813.048} C_VEL
LIN {X 0,Y 458.462,Z 975.994,A -85,B 0,C 180,E1 20810.559,E2 20810.559} C_VEL
